// TwinCAT 3 PLC project MONETRuntime
// ProgramVersion: 3.1.4023.0
// libraries:
//   AstroBROT, * (BROT)
//   Tc2_DataExchange, * (Beckhoff Automation GmbH)
//   Tc2_Math, * (Beckhoff Automation GmbH)
//   Tc2_MC2, * (Beckhoff Automation GmbH)
//   Tc2_MC2_Drive, * (Beckhoff Automation GmbH)
//   Tc2_NC, * (Beckhoff Automation GmbH)
//   Tc2_Standard, * (Beckhoff Automation GmbH)
//   Tc2_System, * (Beckhoff Automation GmbH)
//   Tc2_Utilities, * (Beckhoff Automation GmbH)
//   Tc3_IotBase, * (Beckhoff Automation GmbH)
//   Tc3_Module, * (Beckhoff Automation GmbH)
//   VisuDialogs, * (System)
//   VisuSymbols,3.5.10.0,System
// project tree:
//   DUTs/ E_Blink.TcDUT (not stored), E_Horn.TcDUT (not stored), E_TCSCommand.TcDUT (not stored), E_TCSErrors.TcDUT (not stored), E_TelescopeMode.TcDUT (not stored), ST_InfoDataConnection.TcDUT, ST_InfoDataFB.TcDUT, ST_InfoDataGroup.TcDUT
//   / GlobalTextList.TcGTLO, PlcTask.TcTTO (not stored), Visualization Manager.TcVMO (not stored)
//   GVLs/ GVL_Hydraulics.TcGVL (not stored), GVL_Main.TcGVL, GVL_pendant_control.TcGVL (not stored), GVL_Roof.TcGVL (not stored), GVL_Safety.TcGVL, GVL_Telescope.TcGVL
//   POUs/ AzimuthElevationControl.TcPOU (not stored), CoverControl.TcPOU (not stored), DerotatorControl.TcPOU, ElevationControl.TcPOU (not stored), FocusControl.TcPOU, HydraulicsControl.TcPOU, MAIN.TcPOU, PendantControl.TcPOU, RoofControl.TcPOU (not stored), PowerMonitoring.TcPOU (not stored), SafetyHandling.TcPOU, TelescopeAuxiliary.TcPOU, TelescopeControl.TcPOU
//   POUs/FunctionBlocks/ FB_AstroClock.TcPOU (not stored), FB_Axis2.TcPOU (not stored), FB_BLINK.TcPOU (not stored), FB_ButtonEnable.TcPOU (not stored), FB_Cover.TcPOU (not stored), FB_EventLog.TcPOU (not stored), FB_Horn.TcPOU (not stored), FB_InfluxMessage.TcPOU (not stored), FB_InfoConnection.TcPOU, FB_InfoEStop.TcPOU, FB_InfoGroup.TcPOU, FB_LightTimer.TcPOU (not stored), FB_MQTTCommunication.TcPOU, FB_RFTRIG.TcPOU (not stored), FB_TimeAverage.TcPOU (not stored), FB_Timer.TcPOU (not stored), FB_TONTP.TcPOU (not stored), TelescopeAxisClass.TcPOU (not stored)
//   POUs/Functions/ CT2LST.TcPOU (not stored), F_Azimuthvelocity.TcPOU (not stored), F_DerotatorPosition2.TcPOU (not stored), F_Derotatorvelocity.TcPOU (not stored), F_Elevationvelocity.TcPOU (not stored), F_YREAL.TcPOU (not stored), NCError_TO_STRING.TcPOU (not stored), PointingModelAzimuth.TcPOU (not stored), PointingModelElevation.TcPOU (not stored), Refraction.TcPOU (not stored)
//   VISUs/ Hydraulics.TcVIS (not stored), Safety.TcVIS, Visualization.TcVIS
// real-time tasks:
//   TASK PlcTask: cycle T#10ms, priority 20, ADS port 350
// motion (NC):
//   TASK NC-Task 1 SAF: cycle T#2ms, priority 4, ADS port 501
//   TASK NC-Task 1 SVB: cycle T#10ms, priority 8, ADS port 511
//   AXIS Fokus (id 1)
//     Dynamic: AccelerationMaximum=100, DecelerationMaximum=100, Acceleration=4.5, Deceleration=4.5, Jerk=13.5
//     Velo: RefSearch=0.2, RefSync=0.2, SlowManual=0.1, FastManual=0.5, Maximum=3
//     OtherSettings: AllowMotionCmdToSlave=true, PulseDistancePos=1, PulseDistanceNeg=1
//     encoder EncType=4
//       EncPara: ScaleFactorNumerator=0.001, ScaleFactorDenominator=5, MaxCount=#x0000ffff
//         SoftEndMaxControl: Range=100
//         Inc: RefSoftSyncMask=#x0000ffff
//     drive DrvType=23
//       Analog: VeloReferenz=10.2713178, TorqueSetpointScale=10, ScaleFactorActTorque=0.2
//       TimeComp: TaskDelayCycles=1
//     controller CtrType=1
//       CtrPara: PriorControlFactor=1
//         PID: PosKp=200, CtrlOutputLimit=1
//         Observer: BandWidth=20
//   AXIS Azimuth (id 3)
//     General: UnitName=°
//     Dynamic: AccelerationMaximum=10, DecelerationMaximum=10, Acceleration=10, Deceleration=10, Jerk=4617
//     Velo: RefSearch=10.26, RefSync=10.26, SlowManual=51.3, FastManual=307.8, Fast=1026, Maximum=1026
//     OtherSettings: AllowMotionCmdToSlave=true
//     encoder EncType=8
//       EncPara: ScaleFactorNumerator=360, ScaleFactorDenominator=1048576, MaxCount=#xffffffff
//         SoftEndMinControl: Enable=true
//         SoftEndMaxControl: Enable=true, Range=450
//         Inc: RefPosition=180, RefMode=2
//     drive DrvType=9
//       DrvPara: MaxCount=#xffffffff, DriveControlDWord=#x00030100
//         Analog: VeloReferenz=1128.6, VeloScale=1.02400649589962, TorqueSetpointScale=10, ScaleFactorActTorque=0.1
//         TimeComp: TaskDelayCycles=1
//     controller CtrType=1
//       CtrPara: PriorControlFactor=1
//         PosDiffControl: Range=10
//         Observer: BandWidth=20
//   AXIS Elevation (id 4)
//     General: UnitName=°
//     Dynamic: AccelerationMaximum=10, DecelerationMaximum=10, Acceleration=10, Deceleration=10, Jerk=4617
//     Velo: RefSearch=1, RefSync=1, SlowManual=1, FastManual=3, Fast=1026, Maximum=1026
//     OtherSettings: AllowMotionCmdToSlave=true
//     encoder EncType=8
//       EncPara: ScaleFactorNumerator=360, ScaleFactorDenominator=1048576, MaxCount=#xffffffff
//         SoftEndMinControl: Enable=true
//         SoftEndMaxControl: Enable=true, Range=91
//         Inc: RefPosition=73.9885, RefMode=2
//     drive DrvType=9
//       DrvPara: MaxCount=#xffffffff, DriveControlDWord=#x00030100
//         Analog: VeloReferenz=1128.6, VeloScale=1.02400649589962, TorqueSetpointScale=10, ScaleFactorActTorque=0.1
//         TimeComp: TaskDelayCycles=1
//     controller CtrType=1
//       CtrPara: PriorControlFactor=1
//         PosDiffControl: Range=10
//         Observer: BandWidth=20
//   AXIS Derotator (id 6)
//     General: UnitName=°
//     Dynamic: Acceleration=17.5834, Deceleration=17.5834, Jerk=52.7501
//     Velo: RefSearch=0.117222517903646, RefSync=0.117222517903646, SlowManual=0.586112589518229, FastManual=3.51667553710938, Fast=11.7222517903646, Maximum=11.7223
//     OtherSettings: AllowMotionCmdToSlave=true
//     encoder EncType=8
//       EncPara: ScaleFactorNumerator=0.2, ScaleFactorDenominator=1048576, MaxCount=#xffffffff
//     drive DrvType=9
//       DrvPara: MaxCount=#xffffffff, DriveControlDWord=#x00030100
//         Analog: VeloReferenz=12.894476969401, VeloScale=1.02400649589962, TorqueSetpointScale=10, ScaleFactorActTorque=0.1
//         TimeComp: TaskDelayCycles=1
//     controller CtrType=1
//       CtrPara: PriorControlFactor=1
//         Observer: BandWidth=20
// I/O:
//   DEVICE Device 1 (EtherCAT), AmsNetId 5.131.251.159.2.1
//     Term 21 (EK1200) [EK1200-5000 EtherCAT Power supply (2A E-Bus)]
//       Term 31 (EL1004) [EL1004 4Ch. Dig. Input 24V, 3ms]
//       Temperature IN (EL3202) [EL3202 2Ch. Ana. Input PT100 (RTD)]
//       Brake AzEl (EL2004) [EL2004 4Ch. Dig. Output 24V, 0.5A] // Ch2
//       Safety Logic (EL6910) [EL6910, TwinSAFE PLC]
//       Safety IN (EL1904) [EL1904, 4 Ch. Safety Input 24V, TwinSAFE]
//         modules: Module 1 (FSOES)
//       Safety OUT (EL2904) [EL2904, 4 Ch. Safety Output 24V, 0.5A, TwinSAFE]
//         modules: Module 1 (FSOES), Module 2 (DO)
//       Hydraulics OUT (EL2008) [EL2008 8Ch. Dig. Output 24V, 0.5A] // 1: Start Oil pump. 2: Reset, 3: Start Suction pump, 4: Reset, 5: Start Oil heater, 6: Restart, 7: Brake Focus
//       Hydraulics Focus IN (EL1008) [EL1008 8Ch. Dig. Input 24V, 3ms]
//       Hydraulics IN2 (EL1008) [EL1008 8Ch. Dig. Input 24V, 3ms]
//       Focus Motor (EL7342) [EL7342 2Ch. DC motor output stage (50V, 3.5A)]
//       Mirror Temperature IN (EL3164) [EL3164 4Ch. Ana. Input 0-10V]
//       Power Analysis (EL3483) [EL3483 3Ch. Mains Monitoring]
//       Power (EL9410) [EL9410 E-Bus Power Supplier  (Diagnostics)]
//       Mirror Cover OUT1 (EL2004) [EL2004 4Ch. Dig. Output 24V, 0.5A]
//       Mirror Cover OUT2 (EL2004) [EL2004 4Ch. Dig. Output 24V, 0.5A]
//       Mirror Cover IN (EL1008) [EL1008 8Ch. Dig. Input 24V, 3ms]
//       Front Panel IN (EL1008) [EL1008 8Ch. Dig. Input 24V, 3ms]
//       Front Panel OUT (EL2004) [EL2004 4Ch. Dig. Output 24V, 0.5A]
//       Pendant Control IN (EL1008) [EL1008 8Ch. Dig. Input 24V, 3ms]
//       Pendant Control IN2 (EL1008) [EL1008 8Ch. Dig. Input 24V, 3ms]
//       Pendant Control OUT (EL2008) [EL2008 8Ch. Dig. Output 24V, 0.5A]
//       Cabinet OUT (EL2004) [EL2004 4Ch. Dig. Output 24V, 0.5A]
//       Term 48 (EL9011) [EL9011 End Terminal]
//   DEVICE Device 5 (EtherCAT), AmsNetId 5.131.251.159.6.1
//     Azimuth (AX5125-0000-0214) [AX5125-0000-0214 EtherCAT Drive (SoE, 1 Ch.)]
//       Term 2 (AX5805) [AX5805 (Safety Drive Option)]
//         modules: Module 1 (Safety Process Data, 1 axis), Module 2 (Standard Process Data, 1 axis)
//       Term 7 (EL9011) [EL9011 End Terminal]
//     Elevation (AX5125-0000-0214) [AX5125-0000-0214 EtherCAT Drive (SoE, 1 Ch.)]
//       Term 4 (AX5805) [AX5805 (Safety Drive Option)]
//         modules: Module 1 (Safety Process Data, 1 axis), Module 2 (Standard Process Data, 1 axis)
//       Term 8 (EL9011) [EL9011 End Terminal]
//     Derotator (AX5206-0000-0214) [AX5206-0000-0214 EtherCAT Drive (SoE, 2 Ch.)]
//       Term 6 (AX5805) [AX5805 (Safety Drive Option)]
//         modules: Module 1 (Safety Process Data, 2 axis), Module 2 (Standard Process Data, 2 axis)
//       Term 9 (EL9011) [EL9011 End Terminal]
// variable links:
//   Device 1 (EtherCAT) <-> Device 1 (EtherCAT)/Term 21 (EK1200)/Safety IN (EL1904)
//     Term 21 (EK1200)/Safety Logic (EL6910)/ConnectionInputs/Message_7 TxPDO <-> Module 1 (FSOES)/RxPDO/FSOE
//     Term 21 (EK1200)/Safety Logic (EL6910)/ConnectionOutputs/Message_7 RxPDO <-> Module 1 (FSOES)/TxPDO/FSOE
//   Device 1 (EtherCAT) <-> Device 1 (EtherCAT)/Term 21 (EK1200)/Safety Logic (EL6910)
//     Term 21 (EK1200)/Safety OUT (EL2904)/Module 1 (FSOES)/TxPDO/FSOE <-> ConnectionOutputs/Message_8 RxPDO
//   Device 1 (EtherCAT) <-> Device 1 (EtherCAT)/Term 21 (EK1200)/Safety OUT (EL2904)
//     Term 21 (EK1200)/Safety Logic (EL6910)/ConnectionInputs/Message_8 TxPDO <-> Module 1 (FSOES)/RxPDO/FSOE
//   Device 1 (EtherCAT) <-> Device 5 (EtherCAT)/Azimuth (AX5125-0000-0214)/Term 2 (AX5805)
//     Term 21 (EK1200)/Safety Logic (EL6910)/ConnectionInputs/Message_5 TxPDO <-> Module 1 (Safety Process Data, 1 axis)/Outputs (Controlword)/FSOE
//     Term 21 (EK1200)/Safety Logic (EL6910)/ConnectionOutputs/Message_5 RxPDO <-> Module 1 (Safety Process Data, 1 axis)/Inputs (Statusword)/FSOE
//   Device 1 (EtherCAT) <-> Device 5 (EtherCAT)/Derotator (AX5206-0000-0214)/Term 6 (AX5805)
//     Term 21 (EK1200)/Safety Logic (EL6910)/ConnectionOutputs/Message_17 RxPDO <-> Module 1 (Safety Process Data, 2 axis)/Inputs (Statusword)/FSOE
//   Device 5 (EtherCAT) <-> Device 1 (EtherCAT)/Term 21 (EK1200)/Safety Logic (EL6910)
//     Derotator (AX5206-0000-0214)/Term 6 (AX5805)/Module 1 (Safety Process Data, 2 axis)/Outputs (Controlword)/FSOE <-> ConnectionInputs/Message_17 TxPDO
//     Elevation (AX5125-0000-0214)/Term 4 (AX5805)/Module 1 (Safety Process Data, 1 axis)/Inputs (Statusword)/FSOE <-> ConnectionOutputs/Message_6 RxPDO
//     Elevation (AX5125-0000-0214)/Term 4 (AX5805)/Module 1 (Safety Process Data, 1 axis)/Outputs (Controlword)/FSOE <-> ConnectionInputs/Message_6 TxPDO
//   NC-Task 1 SAF/Axes/Azimuth <-> Device 5 (EtherCAT)/Azimuth (AX5125-0000-0214)
//     Drive/Inputs/In/nDataIn1 <-> AT/Following distance
//     Drive/Inputs/In/nDcOutputTime <-> InfoData/DcOutputShift
//     Drive/Inputs/In/nState1 <-> AT/Drive status word @bit 8
//     Drive/Inputs/In/nState2 <-> AT/Drive status word
//     Drive/Inputs/In/nState4 @bit 1 <-> WcState/InputToggle
//     Drive/Inputs/In/nState4 <-> WcState/WcState
//     Drive/Outputs/Out/nCtrl1 <-> MDT/Master control word @bit 8
//     Drive/Outputs/Out/nDataOut1 <-> MDT/Position command value
//     Enc/Inputs/In/nDataIn1 <-> AT/Position feedback 1 value
//     Enc/Inputs/In/nDataIn3 <-> AT/Probe value 1 positive edge
//     Enc/Inputs/In/nDataIn4 <-> AT/Probe value 1 negative edge
//     Enc/Inputs/In/nDcInputTime <-> InfoData/DcInputShift
//     Enc/Inputs/In/nState4 @bit 1 <-> WcState/InputToggle
//     Enc/Inputs/In/nState4 <-> WcState/WcState
//     Enc/Inputs/In/nState5 <-> AT/Probe 1 positive latched
//     Enc/Inputs/In/nState6 <-> AT/Probe 1 negative latched
//     Enc/Outputs/Out/nCtrl5 <-> MDT/Probe 1 enable
//   NC-Task 1 SAF/Axes/Derotator <-> Device 5 (EtherCAT)/Derotator (AX5206-0000-0214)
//     Drive/Inputs/In/nDataIn1 <-> AT 1/Following distance
//     Drive/Inputs/In/nDcOutputTime <-> InfoData/DcOutputShift
//     Drive/Inputs/In/nState1 <-> AT 1/Drive status word @bit 8
//     Drive/Inputs/In/nState2 <-> AT 1/Drive status word
//     Drive/Inputs/In/nState4 @bit 1 <-> WcState/InputToggle
//     Drive/Inputs/In/nState4 <-> WcState/WcState
//     Drive/Outputs/Out/nCtrl1 <-> MDT 1/Master control word @bit 8
//     Drive/Outputs/Out/nDataOut1 <-> MDT 1/Position command value
//     Enc/Inputs/In/nDataIn1 <-> AT 1/Position feedback 1 value
//     Enc/Inputs/In/nDcInputTime <-> InfoData/DcInputShift
//     Enc/Inputs/In/nState4 @bit 1 <-> WcState/InputToggle
//     Enc/Inputs/In/nState4 <-> WcState/WcState
//   NC-Task 1 SAF/Axes/Elevation <-> Device 5 (EtherCAT)/Elevation (AX5125-0000-0214)
//     Drive/Inputs/In/nDataIn1 <-> AT/Following distance
//     Drive/Inputs/In/nDcOutputTime <-> InfoData/DcOutputShift
//     Drive/Inputs/In/nState1 <-> AT/Drive status word @bit 8
//     Drive/Inputs/In/nState2 <-> AT/Drive status word
//     Drive/Inputs/In/nState4 @bit 1 <-> WcState/InputToggle
//     Drive/Inputs/In/nState4 <-> WcState/WcState
//     Drive/Outputs/Out/nCtrl1 <-> MDT/Master control word @bit 8
//     Drive/Outputs/Out/nDataOut1 <-> MDT/Position command value
//     Enc/Inputs/In/nDataIn1 <-> AT/Position feedback 1 value
//     Enc/Inputs/In/nDataIn3 <-> AT/Probe value 1 positive edge
//     Enc/Inputs/In/nDataIn4 <-> AT/Probe value 1 negative edge
//     Enc/Inputs/In/nDcInputTime <-> InfoData/DcInputShift
//     Enc/Inputs/In/nState4 @bit 1 <-> WcState/InputToggle
//     Enc/Inputs/In/nState4 <-> WcState/WcState
//     Enc/Inputs/In/nState5 <-> AT/Probe 1 positive latched
//     Enc/Inputs/In/nState6 <-> AT/Probe 1 negative latched
//     Enc/Outputs/Out/nCtrl5 <-> MDT/Probe 1 enable
//   NC-Task 1 SAF/Axes/Fokus <-> Device 1 (EtherCAT)/Term 21 (EK1200)/Focus Motor (EL7342)
//     Drive/Inputs/In/nDcOutputTime <-> InfoData/DcOutputShift
//     Drive/Inputs/In/nState1 @bit 3 <-> DCM Status Channel 1/Status/Error
//     Drive/Inputs/In/nState1 @bit 5 <-> DCM Status Channel 1/Status/Moving negative
//     Drive/Inputs/In/nState1 @bit 4 <-> DCM Status Channel 1/Status/Moving positive
//     Drive/Inputs/In/nState1 @bit 1 <-> DCM Status Channel 1/Status/Ready
//     Drive/Inputs/In/nState1 <-> DCM Status Channel 1/Status/Ready to enable
//     Drive/Inputs/In/nState1 @bit 6 <-> DCM Status Channel 1/Status/Torque reduced
//     Drive/Inputs/In/nState1 @bit 2 <-> DCM Status Channel 1/Status/Warning
//     Drive/Inputs/In/nState2 @bit 3 <-> DCM Status Channel 1/Status/Digital input 1
//     Drive/Inputs/In/nState2 @bit 4 <-> DCM Status Channel 1/Status/Digital input 2
//     Drive/Inputs/In/nState2 @bit 5 <-> DCM Status Channel 1/Status/Sync error
//     Drive/Inputs/In/nState2 @bit 7 <-> DCM Status Channel 1/Status/TxPDO Toggle
//     Drive/Inputs/In/nState4 @bit 1 <-> WcState/InputToggle
//     Drive/Inputs/In/nState4 <-> WcState/WcState
//     Drive/Outputs/Out/nCtrl1 <-> DCM Control Channel 1/Control/Enable
//     Drive/Outputs/Out/nCtrl1 @bit 2 <-> DCM Control Channel 1/Control/Reduce torque
//     Drive/Outputs/Out/nCtrl1 @bit 1 <-> DCM Control Channel 1/Control/Reset
//     Drive/Outputs/Out/nCtrl1 @bit 3 <-> DCM Control Channel 1/Control/Threshold active
//     Drive/Outputs/Out/nDataOut2[0] <-> DCM Velocity Channel 1/Velocity
//     Enc/Inputs/In/nDataIn1[0] <-> ENC Status compact Channel 1/Counter value
//     Enc/Inputs/In/nDataIn2[0] <-> ENC Status compact Channel 1/Latch value
//     Enc/Inputs/In/nDcInputTime <-> InfoData/DcInputShift
//     Enc/Inputs/In/nState1 @bit 4 <-> ENC Status compact Channel 1/Status/Counter overflow
//     Enc/Inputs/In/nState1 @bit 3 <-> ENC Status compact Channel 1/Status/Counter underflow
//     Enc/Inputs/In/nState1 @bit 7 <-> ENC Status compact Channel 1/Status/Extrapolation stall
//     Enc/Inputs/In/nState1 @bit 1 <-> ENC Status compact Channel 1/Status/Latch extern valid
//     Enc/Inputs/In/nState1 @bit 2 <-> ENC Status compact Channel 1/Status/Set counter done
//     Enc/Inputs/In/nState2 @bit 4 <-> ENC Status compact Channel 1/Status/Status of extern latch
//     Enc/Inputs/In/nState2 <-> ENC Status compact Channel 1/Status/Status of input A
//     Enc/Inputs/In/nState2 @bit 1 <-> ENC Status compact Channel 1/Status/Status of input B
//     Enc/Inputs/In/nState2 @bit 5 <-> ENC Status compact Channel 1/Status/Sync error
//     Enc/Inputs/In/nState2 @bit 7 <-> ENC Status compact Channel 1/Status/TxPDO Toggle
//     Enc/Inputs/In/nState4 @bit 1 <-> WcState/InputToggle
//     Enc/Inputs/In/nState4 <-> WcState/WcState
//     Enc/Outputs/Out/nCtrl1 @bit 3 <-> ENC Control compact Channel 1/Control/Enable latch extern on negative edge
//     Enc/Outputs/Out/nCtrl1 @bit 1 <-> ENC Control compact Channel 1/Control/Enable latch extern on positive edge
//     Enc/Outputs/Out/nCtrl1 @bit 2 <-> ENC Control compact Channel 1/Control/Set counter
//     Enc/Outputs/Out/nDataOut1[0] <-> ENC Control compact Channel 1/Set counter value
//   MONETRuntime/MONETRuntime Instance <-> Device 1 (EtherCAT)/Term 21 (EK1200)/Brake AzEl (EL2004)
//     PlcTask Outputs/GVL_Telescope.brake_azimuth_eve <-> Channel 2/GVL_Telescope.brake_azimuth_eve
//   MONETRuntime/MONETRuntime Instance <-> Device 1 (EtherCAT)/Term 21 (EK1200)/Front Panel IN (EL1008)
//     PlcTask Inputs/GVL_Main.brake_clearing <-> Channel 5/GVL_Main.key_brake_clearing
//     PlcTask Inputs/GVL_Main.key_switch_remote <-> Channel 4/GVL_Main.key_switch_remote
//     PlcTask Inputs/GVL_Main.reset_switch <-> Channel 3/GVL_Main.reset_switch
//     PlcTask Inputs/GVL_Main.start_switch <-> Channel 1/GVL_Main.start_switch
//     PlcTask Inputs/GVL_Main.stop_switch <-> Channel 2/GVL_Main.stop_switch
//   MONETRuntime/MONETRuntime Instance <-> Device 1 (EtherCAT)/Term 21 (EK1200)/Front Panel OUT (EL2004)
//     PlcTask Outputs/GVL_Main.lamp_error <-> Channel 3/GVL_Main.lamp_error
//     PlcTask Outputs/GVL_Main.lamp_on_manual <-> Channel 2/GVL_Main.lamp_ready
//     PlcTask Outputs/GVL_Main.lamp_power <-> Channel 1/GVL_Main.lamp_power
//   MONETRuntime/MONETRuntime Instance <-> Device 1 (EtherCAT)/Term 21 (EK1200)/Hydraulics Focus IN (EL1008)
//     PlcTask Inputs/GVL_Hydraulics.pump_running <-> Channel 1/GVL_Hydraulics.pump_running
//     PlcTask Inputs/GVL_Hydraulics.suction_running <-> Channel 2/GVL_Hydraulics.suction_running
//     PlcTask Inputs/GVL_Telescope.focus_limit_far <-> Channel 5/GVL_Telescope.focus_limit_far
//     PlcTask Inputs/GVL_Telescope.focus_limit_near <-> Channel 4/GVL_Telescope.focus_limit_near
//   MONETRuntime/MONETRuntime Instance <-> Device 1 (EtherCAT)/Term 21 (EK1200)/Hydraulics IN2 (EL1008)
//     PlcTask Inputs/GVL_Hydraulics.oil_high <-> Channel 2/GVL_Hydraulics.oil_high
//     PlcTask Inputs/GVL_Hydraulics.oil_low <-> Channel 1/GVL_Hydraulics.oil_low
//     PlcTask Inputs/GVL_Hydraulics.oil_overtemperature <-> Channel 4/GVL_Hydraulics.oil_overtemperature
//     PlcTask Inputs/GVL_Hydraulics.oil_pressure_OK <-> Channel 3/GVL_Hydraulics.pressure_OK
//     PlcTask Inputs/GVL_Hydraulics.oil_reserve <-> Channel 8/GVL_Hydraulics.oil_reserve
//     PlcTask Inputs/GVL_Hydraulics.oil_undertemperature <-> Channel 5/GVL_Hydraulics.oil_undertemperature
//     PlcTask Inputs/GVL_Hydraulics.oilfilter_dirty <-> Channel 6/GVL_Hydraulics.oilfilter_dirty
//     PlcTask Inputs/GVL_Hydraulics.oilpan_maximum <-> Channel 7/GVL_Hydraulics.oilpan_maximum
//   MONETRuntime/MONETRuntime Instance <-> Device 1 (EtherCAT)/Term 21 (EK1200)/Hydraulics OUT (EL2008)
//     PlcTask Outputs/GVL_Hydraulics.oil_pump_enable <-> Channel 1/GVL_Hydraulics.oil_pump_enable
//     PlcTask Outputs/GVL_Hydraulics.oil_suction_enable <-> Channel 3/GVL_Hydraulics.oil_suction_enable
//     PlcTask Outputs/GVL_Telescope.focus_unlock <-> Channel 7/GVL_Telescope.focus_unlock
//   MONETRuntime/MONETRuntime Instance <-> Device 1 (EtherCAT)/Term 21 (EK1200)/Mirror Cover IN (EL1008)
//     PlcTask Inputs/GVL_Telescope.cover1_closed <-> Channel 2/GVL_Telescope.cover1_closed
//     PlcTask Inputs/GVL_Telescope.cover2_closed <-> Channel 4/GVL_Telescope.cover2_closed
//     PlcTask Inputs/GVL_Telescope.cover3_closed <-> Channel 6/GVL_Telescope.cover3_closed
//     PlcTask Inputs/GVL_Telescope.cover1_open <-> Channel 1/GVL_Telescope.cover1_open
//     PlcTask Inputs/GVL_Telescope.cover2_open <-> Channel 3/GVL_Telescope.cover2_open
//     PlcTask Inputs/GVL_Telescope.cover3_open <-> Channel 5/GVL_Telescope.cover3_open
//   MONETRuntime/MONETRuntime Instance <-> Device 1 (EtherCAT)/Term 21 (EK1200)/Mirror Cover OUT1 (EL2004)
//     PlcTask Outputs/GVL_Telescope.close_cover1 <-> Channel 2/GVL_Telescope.close_cover1
//     PlcTask Outputs/GVL_Telescope.close_cover2 <-> Channel 4/GVL_Telescope.close_cover2
//     PlcTask Outputs/GVL_Telescope.open_cover1 <-> Channel 1/GVL_Telescope.open_cover1
//     PlcTask Outputs/GVL_Telescope.open_cover2 <-> Channel 3/GVL_Telescope.open_cover2
//   MONETRuntime/MONETRuntime Instance <-> Device 1 (EtherCAT)/Term 21 (EK1200)/Mirror Cover OUT2 (EL2004)
//     PlcTask Outputs/GVL_Telescope.close_cover3 <-> Channel 2/GVL_Telescope.close_cover3
//     PlcTask Outputs/GVL_Telescope.open_cover3 <-> Channel 1/GVL_Telescope.open_cover3
//   MONETRuntime/MONETRuntime Instance <-> Device 1 (EtherCAT)/Term 21 (EK1200)/Mirror Temperature IN (EL3164)
//     PlcTask Inputs/GVL_Telescope.temperature_mirror1 <-> AI Standard Channel 2/Value
//     PlcTask Inputs/GVL_Telescope.temperature_mirror2 <-> AI Standard Channel 1/Value
//   MONETRuntime/MONETRuntime Instance <-> Device 1 (EtherCAT)/Term 21 (EK1200)/Pendant Control IN (EL1008)
//     PlcTask Inputs/GVL_pendant_control.BCD1 <-> Channel 1/GVL_pendant_control.BCD0
//     PlcTask Inputs/GVL_pendant_control.BCD2 <-> Channel 2/GVL_pendant_control.BCD2
//     PlcTask Inputs/GVL_pendant_control.BCD4 <-> Channel 3/GVL_pendant_control.BCD4
//     PlcTask Inputs/GVL_pendant_control.BCD8 <-> Channel 4/GVL_pendant_control.BCD8
//     PlcTask Inputs/GVL_pendant_control.direction_down <-> Channel 7/GVL_pendant_control.direction_down
//     PlcTask Inputs/GVL_pendant_control.direction_up <-> Channel 6/GVL_pendant_control.direction_up
//     PlcTask Inputs/GVL_pendant_control.key_switch <-> Channel 8/GVL_pendant_control.key_switch
//     PlcTask Inputs/GVL_pendant_control.reset_switch <-> Channel 5/GVL_pendant_control.reset_switch
//   MONETRuntime/MONETRuntime Instance <-> Device 1 (EtherCAT)/Term 21 (EK1200)/Pendant Control IN2 (EL1008)
//     PlcTask Inputs/GVL_pendant_control.direction_left <-> Channel 2/GVL_pendant_control.direction_left
//     PlcTask Inputs/GVL_pendant_control.direction_right <-> Channel 3/GVL_pendant_control.direction_right
//     PlcTask Inputs/GVL_pendant_control.start_switch <-> Channel 1/GVL_pendant_control.start_switch
//   MONETRuntime/MONETRuntime Instance <-> Device 1 (EtherCAT)/Term 21 (EK1200)/Pendant Control OUT (EL2008)
//     PlcTask Outputs/GVL_pendant_control.lamp_down <-> Channel 2/GVL_pendant_control.lamp_down
//     PlcTask Outputs/GVL_pendant_control.lamp_error <-> Channel 5/GVL_pendant_control.lamp_error
//     PlcTask Outputs/GVL_pendant_control.lamp_left <-> Channel 4/GVL_pendant_control.lamp_left
//     PlcTask Outputs/GVL_pendant_control.lamp_right <-> Channel 3/GVL_pendant_control.lamp_right
//     PlcTask Outputs/GVL_pendant_control.lamp_up <-> Channel 1/GVL_pendant_control.lamp_up
//   MONETRuntime/MONETRuntime Instance <-> Device 1 (EtherCAT)/Term 21 (EK1200)/Safety Logic (EL6910)
//     PlcTask Inputs/GVL_Telescope.Azimuth_sto <-> StandardInputs/Standard Out Var 18
//     PlcTask Inputs/GVL_Telescope.Derotator_sto <-> StandardInputs/Standard Out Var 20
//     PlcTask Inputs/GVL_Telescope.Elevation_sto <-> StandardInputs/Standard Out Var 19
//     PlcTask Inputs/SafetyHandling.stInfoEStop1 <-> Function Block Info Data/TwinSafeGroup1.Network1.FBEstop1 Info Data
//     PlcTask Inputs/SafetyHandling.stInfoGroup1 <-> TwinSAFE Group Info Data/TwinSafeGroup1 Info Data
//     PlcTask Inputs/SafetyHandling.stInfoSafetyIn <-> Connection Info Data/Message_8 Info Data
//     PlcTask Inputs/SafetyHandling.stInfoSafetyOut <-> Connection Info Data/Message_7 Info Data
//     PlcTask Outputs/GVL_Safety.ErrAck <-> StandardOutputs/Standard In Var 1
//     PlcTask Outputs/GVL_Safety.Reset_STO_Azimuth <-> StandardOutputs/Standard In Var 25
//     PlcTask Outputs/GVL_Safety.Reset_STO_Derotator <-> StandardOutputs/Standard In Var 22
//     PlcTask Outputs/GVL_Safety.Reset_STO_Elevation <-> StandardOutputs/Standard In Var 26
//     PlcTask Outputs/GVL_Safety.Restart <-> StandardOutputs/Standard In Var 3
//     PlcTask Outputs/GVL_Safety.Run <-> StandardOutputs/Standard In Var 2
//   MONETRuntime/MONETRuntime Instance <-> Device 1 (EtherCAT)/Term 21 (EK1200)/Temperature IN (EL3202)
//     PlcTask Inputs/GVL_Main.main_cabinet_temperature <-> RTD Inputs Channel 1/Value

// ---- DUTs/ST_InfoDataConnection.TcDUT
TYPE ST_InfoDataConnection :
STRUCT
	usiMapState	:USINT;
	usiMapDiag	:USINT;
	bySignal	:BYTE;
END_STRUCT
END_TYPE

// ---- DUTs/ST_InfoDataFB.TcDUT
TYPE ST_InfoDataFB :
STRUCT
	usiMapState	:USINT;
	uiMapDiag	:USINT;
	usiDummy	:USINT;
END_STRUCT
END_TYPE

// ---- DUTs/ST_InfoDataGroup.TcDUT
TYPE ST_InfoDataGroup :
STRUCT
	usiMapState	:USINT;
	usiMapDiag	:USINT;	
END_STRUCT
END_TYPE

// ---- GVLs/GVL_Main.TcGVL
{attribute 'qualified_only'}
//TODO update to current RoboTel IOs
VAR_GLOBAL
	//DIN1 0.0
	//phase_available		AT%I*: BOOL;
	//not implemented on RoboTel
	//key_switch			AT%I*: BOOL;
	//DIN3 0.2
	key_switch_remote	AT%I*: BOOL;
	//DIN4 0.3
	start_switch		AT%I*: BOOL;
	//DIN5 0.4
	stop_switch			AT%I*: BOOL;
	//DIN8 0.7
	reset_switch		AT%I*: BOOL;
	
	//BT1
	main_cabinet_temperature	AT%I*: INT;
	//DIN15 1.6
	brake_clearing		AT%I*: BOOL;
	
	//DOUT1 0.0
	lamp_power			AT%Q*: BOOL;
	//DOUT2 0.1
	lamp_on_manual			AT%Q*: BOOL;
	//DOUT3 0.2
	lamp_error			AT%Q*: BOOL;
	
	isRoboTel:		BOOL;
	(*
	NeutralCurrentGuardWarning		AT%I*:	BOOL;
	NeutralCurrentGuarError			AT%I*:	BOOL;
	ActivePowerGuardWarning			AT%I*:	BOOL;
	ActivePowerGuardError			AT%I*:	BOOL;
	ApparentPowerGuardWarning		AT%I*:	BOOL;
	ApparentPowerGuardError			AT%I*:	BOOL;
	*)
	//ActivePower						AT%I*:	REAL;
	//ActiveEnergy					AT%I*:	LINT;
	//NeutralLineCurrent				AT%I*:	REAL;
END_VAR

// ---- GVLs/GVL_Safety.TcGVL
{attribute 'qualified_only'}
VAR_GLOBAL
	// Safety Error Condition
	Error		AT%I*:	BOOL;
	// Run/Stop Safety
	Run			AT%Q*:	BOOL;
	// Restart Safety
	Restart		AT%Q*:	BOOL;
	// Error Acknowledgement 
	ErrAck		AT%Q*:	BOOL;
	// Stop signal coming from Safety
	// Stop		AT%I*:	BOOL;
	// state variable
	State		AT%I*:	USINT;
	
	Reset_STO_Azimuth		AT%Q*: BOOL;
	Reset_STO_Elevation		AT%Q*: BOOL;
	Reset_STO_Derotator		AT%Q*: BOOL;
END_VAR

// ---- GVLs/GVL_Telescope.TcGVL
{attribute 'qualified_only'}
VAR_GLOBAL
	// BT9 mirror
	temperature_mirror2		AT%I*: INT;
	// BT10
	temperature_mirror1		AT%I*: INT;

	//DOUT6 0.5
	brake_azimuth_eve	AT%Q*: BOOL;
	
	// DIN28 3.3 (absolute)
	azimut_limit_switch	AT%I*: BOOL;
	// DIN29 3.4
	focus_limit_near	AT%I*: BOOL;
	// DIN30 3.5
	focus_limit_far		AT%I*: BOOL;
	
	// DIN33 4.0
	cover1_open		AT%I*: BOOL;
	// DIN34 4.1
	cover1_closed	AT%I*: BOOL;
	// DIN35 4.2
	cover2_open		AT%I*: BOOL;
	// DIN36 4.3
	cover2_closed	AT%I*: BOOL;
	// DIN37 4.4
	cover3_open		AT%I*: BOOL;
	// DIN38 4.5
	cover3_closed	AT%I*: BOOL;

	//DOUT14 1.5
	focus_unlock		AT%Q*: BOOL;
	//Horn 4.7
	horn			AT%Q*: BOOL;
	
	// digitale inputs der Endlagen
	Derotator_inputs		AT%I*: WORD;
	// diagnostic number
	Derotator_diagnostic	AT%I*: UDINT;
	// derotator torque feedback
	Derotator_torque		AT%I*: INT;
	// STO
	Derotator_sto			AT%I*: BOOL;
	
	// digital inputs for limit switches
	Elevation_inputs		AT%I*: WORD;
	// diagnostic number
	Elevation_diagnostic	AT%I*: UDINT;
	// torque feedback
	Elevation_torque		AT%I*: INT;
	// STO
	Elevation_sto			AT%I*: BOOL;
	
	// digital inputs for limit switches
	Azimuth_inputs			AT%I*: WORD;
	// diagnostic number
	Azimuth_diagnostic		AT%I*: UDINT;
	// torque feedback
	Azimuth_torque			AT%I*: INT;
	// STO
	Azimuth_sto				AT%I*: BOOL;	
	
	// Zyklisches Interface zwischen NC und Achse
	AzimuthAxisRef: 	AXIS_REF;
	ElevationAxisRef: 	AXIS_REF;
	DerotatorAxisRef: 	AXIS_REF;
 	// Motor1 Channel 1
	FocusAxisRef:		AXIS_REF;
	
	//nasmyth_left	AT%Q*: BOOL;
	//nasmyth_right	AT%Q*: BOOL;
	open_cover1		AT%Q*: BOOL;
	close_cover1	AT%Q*: BOOL;
	open_cover2		AT%Q*: BOOL;
	close_cover2	AT%Q*: BOOL;
	open_cover3		AT%Q*: BOOL;
	close_cover3	AT%Q*: BOOL;
	
	
END_VAR

// ---- POUs/DerotatorControl.TcPOU
PROGRAM DerotatorControl
VAR_INPUT
	// enable the derotator
	enable:		BOOL;
	// reset an error
	reset:		BOOL;
	// decrease derotator angle
	left:		BOOL;
	// increase derotator angle
	right:		BOOL;
	// set the absolute position
	position:	LREAL;
	// derotator velocity
	Velocity:	LREAL := 10.0;
	// move to given position
	MoveAxis: 	BOOL;
	// calibrate the axis
	HomeAxis:	BOOL;
	// tracking flag
	Tracking:	BOOL;
	// stop the Axis
	StopAxis:	BOOL;
	// diagnostic error code reset
	bSoEReset: 			BOOL;
END_VAR
VAR_OUTPUT
	// error flag
	Error:				BOOL;
	// nc error id
	ErrorID:			UDINT;
	// actual position of the derotator
	actual_position:	LREAL;
	// calibrated flag
	Calibrated:			BOOL;
	// axis ready flag
	Ready:				BOOL;
	// position to move the axis to
	slewtime: 			LREAL;
END_VAR
VAR
	// trigger for the torque error
	TorqueError:		TON := (PT := T#3S);
	// axis function block
	DerotatorAxis:		FB_Axis2;
	
	DerotatorEvent:		FB_EventLog;
	// torque warning event
	TorqueWarning:		FB_EventLog;
	// torque calibration event
	CalibrationEvent:	FB_EventLog;
	// diagnostic low-level event
	DerotatorDiagnosticEvent: FB_EventLog;
	// percentage of the derotator torque
	derotator_torque:	REAL;
	// read slewtime
	ReadParameter:		MC_ReadParameter;
	fbSoEReset: 		FB_SoEReset;
	DiagnosticError:	BOOL;
END_VAR
VAR CONSTANT
	// current position of the calibration cam. Apply an offset here if necessary
	calibration_position:	LREAL := 438.4623; // calibration in positive direction (was 460.0)
END_VAR

(*
Selection 6
Homing in Endlage:

https://infosys.beckhoff.com/index.php?content=../content/1031/ax5000_usermanual/html/ax5000_homing_hardware_end_position.htm&id=12221
NC-Interface:
PlcToNc-Achsinterface, Bit 8 namens AcceptBlockedDriveSignal im nDeCtrlDWord

SPS-Interface:
TcNc-Lib, siehe SPS-Funktion AxisSetAcceptBlockedDriveSignal in der TwinCAT  PLC Library: NC.
*)

position := LIMIT(-70, position, 380);

IF enable AND NOT DerotatorAxis.Calibrated THEN
	HomeAxis := TRUE;
END_IF

IF DerotatorAxis.Calibrated THEN
	HomeAxis := FALSE;
	Calibrated := DerotatorAxis.Calibrated;
END_IF
	
IF HomeAxis THEN
	position := calibration_position;
END_IF

DeRotatorAxis(
	enable := 			enable,
	Reset := 			Reset,
	MoveAxis :=			MoveAxis,
	HomeAxis :=			HomeAxis,
	StopAxis :=			StopAxis,
	HomingMode :=		MC_ForceCalibration,
	Position := 		position, 
	Velocity :=			Velocity,
	Enable_Positive := 	NOT GVL_Telescope.Derotator_inputs.0,
	Enable_Negative := 	NOT GVL_Telescope.Derotator_inputs.1,
	Jog_Forward := 		right,
	Jog_Backwards := 	left,
	bCalibrationCam :=	GVL_Telescope.Derotator_inputs.0,
	isModuloAxis :=		FALSE,
	Tracking :=			Tracking,
	ActualPosition => 	actual_position,
	Error => 			Error,
	ErrorID => 			ErrorID,
	AxisRef :=			GVL_Telescope.DerotatorAxisRef);
	
IF DeRotatorAxis.MoveDone OR Reset OR Error THEN
	MoveAxis := FALSE;
END_IF

IF DeRotatorAxis.HomeDone OR Reset OR Error THEN
	HomeAxis := FALSE;
END_IF
	
IF DeRotatorAxis.ResetDone THEN
	reset := FALSE;
END_IF

IF DeRotatorAxis.StopDone THEN
	StopAxis := FALSE;
END_IF

DiagnosticError := FALSE;
IF GVL_Telescope.Derotator_diagnostic < 16#D012 AND GVL_Telescope.Derotator_diagnostic > 16#D014 THEN
	DiagnosticError := TRUE;
	ErrorID := GVL_Telescope.Derotator_diagnostic;
	bSoeReset := reset;
END_IF

Ready := DeRotatorAxis.Ready;

ReadParameter(	Axis := GVL_Telescope.DerotatorAxisRef, 
				Enable := DeRotatorAxis.InMotion, 
				ParameterNumber := MC_AxisParameter.AxisRemainingTimeToGo, 
				ReadMode := E_ReadMode.READMODE_CYCLIC);
				
IF ReadParameter.Valid THEN
	slewtime := ReadParameter.Value;
END_IF

IF bSoEReset THEN
	fbSoEReset(
		Axis := GVL_Telescope.DerotatorAxisRef,
		Execute := TRUE,
		Timeout := DEFAULT_ADS_TIMEOUT);
 	IF NOT fbSoEReset.Busy THEN
		fbSoEReset(Axis := GVL_Telescope.DerotatorAxisRef, Execute := FALSE);
		bSoEReset := FALSE;
		Reset := TRUE;
	END_IF
END_IF

derotator_torque := GVL_Telescope.Derotator_torque / 10.0;

TorqueError(IN := ABS(derotator_torque) > 12.0);

DerotatorEvent(	
	Trigger := 		Error, 
	Level := 		ADSLOG_MSGTYPE_ERROR,
	FormatString :=	'Derotator Axis Error: %s',
	OnMessage := 	NCError_TO_STRING(ErrorID),
	OffMEssage := 	'OK',
	OffLevel := 	ADSLOG_MSGTYPE_HINT);
	
DerotatorDiagnosticEvent(	
	Trigger := 		DiagnosticError, 
	Level := 		ADSLOG_MSGTYPE_ERROR,
	FormatString :=	'Derotator Axis Diagnostic Error: %s',
	OnMessage := 	NCError_TO_STRING(GVL_Telescope.Derotator_diagnostic));
	
TorqueWarning(	
	Trigger := 		TorqueError.Q, 
	Level := 		ADSLOG_MSGTYPE_WARN,
	FormatString :=	'%s',
	OnMessage := 	'Derotator torque is high.');

CalibrationEvent(	
	Trigger := 		Calibrated, 
	Level := 		ADSLOG_MSGTYPE_HINT,
	OnMessage := 	'Derotator is calibrated.');

END_PROGRAM

// ---- POUs/FocusControl.TcPOU
PROGRAM FocusControl
VAR_INPUT
	// enable the axis
	enable: BOOL;
	// Move M2 closer to M1
	inward: 	BOOL;
	// Move M2 away from M1
	outward: 	BOOL;	
	// reset the axis(-error)
	reset: 		BOOL;
	// move the axis to new position
	MoveAxis:	BOOL;
	// calibrate the focus axis
	HomeAxis:	BOOL;
	// focus position in millimeters
	position: 		LREAL;
END_VAR

VAR_OUTPUT
	// true if absolute calibration
	Calibrated:	BOOL;
	// true if error
	Error: 		BOOL;
	// ID of NC axis error
	ErrorID:	UDINT;
	// ready signal = drive ready + standstill
	Ready:	BOOL;
END_VAR

VAR
	FocusDelay:			TON;
	BrakeDelay:			TON;
	FocusAxis:			FB_Axis2;
	actual_position:	LREAL;
	// manual override to unlock the focus
	FocusUnlock:		BOOL;
	FocusUnlocked:		BOOL;
	MQTTTimer : 		TON := (PT:=T#5S);
	//getlastposition:	BOOL := TRUE;
	FocusAxisEvent:		FB_EventLog;
	CalibrationEvent:	FB_EventLog;
	HomingMode: 		MC_HOMINGMODE := 		MC_DefaultHoming;
	SetPosition:		MC_SetPosition;
END_VAR

VAR CONSTANT
	// reference position for homing
	homing_position:		LREAL := 92.8936; // 106.5936 - 13.7000
	tolerance:				LREAL := 0.005;
END_VAR
VAR PERSISTENT
	last_position:		LREAL := -1.0;
END_VAR

(*
Focus Control Unit
spindle gear: 5mm
brake: 86 61103H00 Var. 0005 Index C; 24VDC geglattet 0,25 A P1672/R7
motor: Faulhaber ; Schönaich ; 3557K024CR; 454  431 ; Made in germany ==> 5300 rpm
gear: Faulhaber ; MINIMOTOR SA ; swiss made ; 38/1S  43:1 ; 033896  503
Focus is locked by default
70,8W; 0,100A no load current; 2,0 Terminal resistance; 1,950A max Current 
*)
position := LIMIT(5.0, position, 95.0);

GVL_Telescope.focus_unlock := FocusUnlock OR enable;

// wait until the focus is unlocked for n milliseconds
FocusDelay(IN := GVL_Telescope.focus_unlock, PT := T#500MS, Q => FocusUnlocked);
// wait for brake until we are at rest
BrakeDelay(IN := NOT FocusAxis.Busy AND FocusAxis.StandStill, PT := T#4000MS);

// if we are on automatic mode then position the focus
IF Pendantcontrol.telescope_mode = E_TelescopeMode.automatic AND NOT FocusUnlock THEN
	IF FocusAxis.Calibrated THEN
		IF ABS(position - actual_position) > tolerance THEN
			IF FocusAxis.Ready THEN
				MoveAxis := TRUE;
			ELSE
				Enable := TRUE;
			END_IF
		END_IF
		// disable the drive and lock the brake, if we stand for more than n seconds
		IF BrakeDelay.Q THEN
			Enable := FALSE;
		END_IF
		// store actual position, if we are calibrated and locked
		IF NOT GVL_Telescope.focus_unlock THEN
			last_position := actual_position;
		END_IF
	ELSE // not calibrated
		IF FocusAxis.Ready THEN
			HomeAxis := TRUE;
		END_IF
	END_IF
END_IF

IF HomeAxis THEN
	IF last_position > 0.0 THEN
		HomingMode := MC_ForceCalibration; // MC_Direct
		position := last_position;
		SetPosition.Execute := TRUE;
	ELSE
		HomingMode := MC_DefaultHoming;
		position := homing_position;
		SetPosition.Execute := FALSE;
	END_IF
ELSE
	SetPosition.Execute := FALSE;	
END_IF

// deactivate limit switches on homing
MC_SetAcceptBlockedDriveSignal(
	Axis := GVL_Telescope.FocusAxisRef, 
	Enable := HomeAxis);
SetPosition(
	Axis := GVL_Telescope.FocusAxisRef, 
	Position := last_position);
	
	
FocusAxis(	
	Enable := 			FocusUnlocked,
	Reset := 			reset,
	MoveAxis := 		MoveAxis AND FocusUnlocked,
	HomeAxis :=			HomeAxis AND FocusUnlocked,
	HomingMode :=		HomingMode,
	Position := 		position,
	Velocity :=			1.0,
	Enable_Positive := 	NOT GVL_Telescope.focus_limit_far OR HomeAxis,
	Enable_Negative := 	NOT GVL_Telescope.focus_limit_near,
	Jog_Forward :=		outward AND FocusUnlocked,
	Jog_Backwards := 	inward AND FocusUnlocked,
	bCalibrationCam :=  GVL_Telescope.focus_limit_far,
	ActualPosition => 	actual_position,
	Error =>			error,
	ErrorID =>			ErrorID,
	AxisRef :=			GVL_Telescope.FocusAxisRef);	

IF FocusAxis.MoveDone THEN
	MoveAxis := FALSE;
END_IF

IF FocusAxis.HomeDone THEN
	HomeAxis := FALSE;
	Enable := FALSE;
	last_position := position;
END_IF
	
IF FocusAxis.ResetDone THEN
	reset := FALSE;
END_IF

IF FocusAxis.Calibrated OR Error THEN
	HomeAxis := FALSE;
END_IF

IF Error THEN
	last_position := -1.0;
	//FocusAxis.Calibrated := FALSE;
	Calibrated := FALSE;
END_IF

Calibrated := FocusAxis.Calibrated;

Ready := FocusAxis.Ready AND FocusAxis.StandStill OR NOT GVL_Telescope.focus_unlock;

MQTTTimer(IN:=TRUE);
IF MQTTTimer.Q THEN // publish new payload every second
	MQTTTimer(IN:=FALSE);
	MAIN.MQTTClient.Publish('telescope', 'dome', 'FocusPosition', LREAL_TO_FMTSTR(actual_position, 5, TRUE));
	MAIN.MQTTClient.Publish('telescope', 'dome', 'FocusCalibrated', BOOL_TO_STRING(Calibrated));	
	MAIN.MQTTClient.Publish('telescope', 'dome', 'FocusReady', BOOL_TO_STRING(Ready));	
END_IF

FocusAxisEvent(	
	Trigger := 		FocusAxis.Error, 
	Level := 		ADSLOG_MSGTYPE_ERROR,
	FormatString :=	'Focus Axis Error: %s',
	OnMessage := 	NCError_TO_STRING(ErrorID),
	OffMEssage := 	'OK',
	OffLevel := 	ADSLOG_MSGTYPE_HINT);

CalibrationEvent(
	Trigger :=	Calibrated,
	Level :=	ADSLOG_MSGTYPE_HINT,
	OnMessage := 'Focus is calibrated.'
	);

END_PROGRAM

// ---- POUs/PendantControl.TcPOU
PROGRAM PendantControl
VAR
	// program selection of the pendant control
	Selection:	UINT;
	// error on the pendant control
	Error:		BOOL;
	// manual switch
	manual:		BOOL;
	//enable button
	enable:		BOOL;
	//reset button
	reset:		BOOL;
	// up button
	up:			BOOL;
	// down button
	down:		BOOL;
	// left button
	left:		BOOL;
	// right button
	right:		BOOL;
	lamp_left:		BOOL;
	lamp_right:		BOOL;
	lamp_up:		BOOL;
	lamp_down:		BOOL;
	lamp_error:		BOOL;
	horn:			BOOL;
	FocusEnable: 		FB_ButtonEnable;
	DerotatorEnable:	FB_ButtonEnable;
	ElevationEnable: 	FB_ButtonEnable;
	AzimuthEnable: 		FB_ButtonEnable;
	TelescopeControlEnable: 	FB_ButtonEnable;
	HydraulicsEnable: 	FB_ButtonEnable;
	TrackingEnable:			FB_ButtonEnable;
	ResetDelay:	TON;
	TwinCATRestart: TC_Restart;
	up_trigger:	R_TRIG;
	down_trigger:	R_TRIG;	
	// manual or automatic operation of the telescope
	telescope_mode : E_TelescopeMode;	
END_VAR

(* 
This program is responsible for the manual control of the telescope.
all movable parts can be controlled from here. This is mainly for testing and
maintenance.
WARNING! Some of the safety routines are disabled, when operating the telescope manually.
*)
// calculate the value of the selector
Selection := 1*BOOL_TO_UINT(GVL_pendant_control.BCD1) + 
			 2*BOOL_TO_UINT(GVL_pendant_control.BCD2) + 
			 4*BOOL_TO_UINT(GVL_pendant_control.BCD4) +
			 8*BOOL_TO_UINT(GVL_pendant_control.BCD8);

// detect disconnection of the manual controls (should also trigger emergency stop).			 
Error := (Selection = 0);

// disable all the lamps
lamp_left := FALSE;
lamp_right := FALSE;
lamp_up := FALSE;
lamp_down := FALSE;
horn := FALSE;

// clooect the state of all buttons
manual := GVL_pendant_control.key_switch;
enable := GVL_pendant_control.start_switch;
reset := GVL_pendant_control.reset_switch;
up := GVL_pendant_control.direction_up;
down := GVL_pendant_control.direction_down;
left := GVL_pendant_control.direction_left;
right := GVL_pendant_control.direction_right;

up_trigger(CLK := up);
down_trigger(CLK := down);
//R_Enable(CLK := enable);
// the error lamp is the same as the error lamp of the main panel
lamp_error := GVL_Main.lamp_error;
CoverControl.active_cover := 0;


// determine the operation of the telescope based on the switch set
IF manual THEN
	telescope_mode := E_TelescopeMode.manual;
ELSE
	telescope_mode := E_TelescopeMode.automatic;
END_IF

// enable only the selected item and connect lamps and buttons accordingly
CASE Selection OF
	1:	// reserved for Cover1 control
		lamp_up := GVL_Telescope.cover1_open;
		lamp_down := GVL_Telescope.cover1_closed;
		IF manual THEN
			//CoverEnable(SET := enable, Q := CoverControl.enable);
			//CoverControl.active_cover := 1;
			//CoverControl.reset := reset;
			GVL_Telescope.open_cover1 := up AND GVL_Telescope.cover1_open;
			GVL_Telescope.close_cover1 := down AND GVL_Telescope.cover1_closed;
			lamp_error := CoverControl.Cover1_Error;	
		ELSE
			IF down THEN 
				CoverControl.close := TRUE;
			END_IF
			IF up THEN
				CoverControl.open := TRUE;
			END_IF		
		END_IF

	2: // Cover2 control
		lamp_up := GVL_Telescope.cover2_open;
		lamp_down := GVL_Telescope.cover2_closed;
		IF manual THEN
			//CoverEnable(SET := enable, Q := CoverControl.enable);
			//CoverControl.active_cover := 2;
			GVL_Telescope.open_cover2 := up AND GVL_Telescope.cover2_open;
			GVL_Telescope.close_cover2 := down AND GVL_Telescope.cover2_closed;
			lamp_error := CoverControl.Cover2_Error;
		ELSE
			IF down THEN 
				CoverControl.close := TRUE;
			END_IF
			IF up THEN
				CoverControl.open := TRUE;
			END_IF		
		END_IF
 	
	3:  // Cover3 control
		lamp_up := GVL_Telescope.cover3_open;
		lamp_down := GVL_Telescope.cover3_closed;
		IF manual THEN
			//CoverEnable(SET := enable, Q := CoverControl.enable);
			//CoverControl.active_cover := 3;
			GVL_Telescope.open_cover3 := up AND GVL_Telescope.cover3_open;
			GVL_Telescope.close_cover3 := down AND GVL_Telescope.cover3_closed;
			//CoverControl.reset := reset;
			lamp_error := CoverControl.Cover3_Error;
		ELSE
			IF down THEN 
				CoverControl.close := TRUE;
			END_IF
			IF up THEN
				CoverControl.open := TRUE;
			END_IF		
		END_IF
		
	4:	// Nasmyth / mirror M3 control
		
	5:	// Focus Control
		lamp_up := FocusControl.Ready AND NOT GVL_Telescope.focus_limit_far;
		lamp_down := FocusControl.Ready AND NOT GVL_Telescope.focus_limit_near;
		IF manual THEN
			FocusEnable(SET := enable, Q := FocusControl.enable);
			FocusControl.outward := up;
			FocusControl.inward := down;
			Focuscontrol.reset := reset;
			lamp_error := FocusControl.error;
		END_IF
							
	6:	// Derotator control
		lamp_left := DerotatorControl.Ready AND NOT GVL_Telescope.Derotator_inputs.1;
		lamp_right :=DerotatorControl.Ready AND NOT GVL_Telescope.Derotator_inputs.0;
		IF manual THEN
			DerotatorEnable(SET := enable, Q := DerotatorControl.enable);
			DerotatorControl.left := left AND NOT GVL_Telescope.Derotator_inputs.1;
			DerotatorControl.right := right AND NOT GVL_Telescope.Derotator_inputs.0;
			DerotatorControl.reset := reset;
			lamp_error := DerotatorControl.Error;
		END_IF
							
	7:	// Elevation Control
		
		ElevationControl.up := up AND GVL_Telescope.Elevation_inputs.0;
		ElevationControl.down := down AND GVL_Telescope.Elevation_inputs.1;
		IF manual THEN
			ElevationEnable(
				SET := enable, 
				Q := ElevationControl.enable);	
		END_IF
		ElevationControl.reset := reset;
		lamp_up := GVL_Telescope.Elevation_inputs.0;
		lamp_down := GVL_Telescope.Elevation_inputs.1;
		lamp_error := ElevationControl.error;
		
	8:	// Azimuth Control
		lamp_left := GVL_Telescope.Azimuth_inputs.0; // NOT GVL_Telescope.azimut_limit_switch;
		lamp_right := GVL_Telescope.Azimuth_inputs.1; // NOT GVL_Telescope.azimut_limit_switch;
		AzimuthElevationControl.left := left AND GVL_Telescope.Azimuth_inputs.0;
		AzimuthElevationControl.right := right AND GVL_Telescope.Azimuth_inputs.1;
		AzimuthElevationControl.reset := reset;
		IF manual THEN
			AzimuthEnable(
				SET := enable, 
				Q := AzimuthElevationControl.enable);
			lamp_error := AzimuthElevationControl.error;
		END_IF
		
	9: 	// Dome control
		
	10:	// FilterWheel control
		
	11: lamp_up := ElevationControl.elevation_torque > 0.0;
		lamp_down := ElevationControl.elevation_torque < 0.0;
		
	12:	// manual Telescope Control
		IF manual THEN
			lamp_up := TelescopeControl.power;
			lamp_down := TelescopeControl.power;
			lamp_left := TelescopeControl.power;
			lamp_right := TelescopeControl.power;
	
			TelescopeControl.gohome := down;
			TelescopeControl.park := up;
			TelescopeControl.goto := right;
			TrackingEnable(SET := enable, 
							RESET := reset, 
							Q := TelescopeControl.track);
			TelescopeControl.reset := reset;
			Telescopecontrol.stop := left;	
			lamp_error := Telescopecontrol.error;
		END_IF
		
	13: // Telescope Control
		TelescopeControlEnable(
			SET := enable, 
			Q := TelescopeControl.power);
		TelescopeControl.reset := reset;
		IF manual THEN
			lamp_up := GVL_Telescope.Elevation_inputs.0;
			lamp_down := GVL_Telescope.Elevation_inputs.1;
			lamp_left := GVL_Telescope.Azimuth_inputs.0;
			lamp_right := GVL_Telescope.Azimuth_inputs.1;
			ElevationControl.up := up AND GVL_Telescope.Elevation_inputs.0;
			ElevationControl.down := down AND GVL_Telescope.Elevation_inputs.1;
			AzimuthElevationControl.left := left AND GVL_Telescope.Azimuth_inputs.0;
			AzimuthElevationControl.right := right AND GVL_Telescope.Azimuth_inputs.1;
			TelescopeControl.rightascension := TelescopeControl.rightascension_calc;
			TelescopeControl.declination := TelescopeControl.declination_calc;
		ELSE
			lamp_up := ElevationControl.enable;
			lamp_down := ElevationControl.enable;
			lamp_left := AzimuthElevationControl.enable;
			lamp_right := AzimuthElevationControl.enable;
			IF up THEN 
				Telescopecontrol.elevation_offset := Telescopecontrol.elevation_offset + 10.0/3600.0; 
			ELSIF down THEN 
				Telescopecontrol.elevation_offset := Telescopecontrol.elevation_offset - 10.0/3600.0; 
			END_IF;
			IF left THEN 
				Telescopecontrol.azimuth_offset := Telescopecontrol.azimuth_offset - 10.0/3600.0; 
			ELSIF right THEN 
				Telescopecontrol.azimuth_offset := Telescopecontrol.azimuth_offset + 10.0/3600.0; 
			END_IF;
		END_IF
		ResetDelay(IN := reset, PT := T#3S);
		// wait for suction pump to stop
		TwinCATRestart(NETID := '', RESTART := ResetDelay.Q AND NOT HydraulicsControl.suction_running, TMOUT := T#60S);
	
	14: horn := manual;
		lamp_up := manual;
		lamp_down := manual;
		lamp_left := manual;
		lamp_right := manual;
	
	15:	// Hydraulics control
		lamp_up := HydraulicsControl.oil_pressure_OK AND Hydraulicscontrol.brake_closed;
		lamp_down := HydraulicsControl.oil_pressure_OK AND Hydraulicscontrol.brake_open;
		lamp_left := HydraulicsControl.pump_running;
		lamp_right := HydraulicsControl.suction_running;
		IF manual THEN
			HydraulicsEnable(
				SET := enable, 
				Q := Hydraulicscontrol.enable);
			Hydraulicscontrol.reset := reset;
			
			IF up THEN
				Hydraulicscontrol.open_brake();
			END_IF
			IF down THEN
				Hydraulicscontrol.close_brake();
			END_IF
			Hydraulicscontrol.suction_manual := right;
			Hydraulicscontrol.pump_manual_stop := left;
			lamp_error := HydraulicsControl.error;
		END_IF
END_CASE

// set all the lamps
GVL_pendant_control.lamp_left := lamp_left;
GVL_pendant_control.lamp_right := lamp_right;
GVL_pendant_control.lamp_up := lamp_up;
GVL_pendant_control.lamp_down := lamp_down;
GVL_pendant_control.lamp_error := lamp_error;

END_PROGRAM

// ---- POUs/TelescopeControl.TcPOU
PROGRAM TelescopeControl
VAR_INPUT
(*
TCS interface section
see https://gitlab.aip.de/bmk10k/telescope_firmware/snippets/5
*)
	
	// boolean, true: Power on, false: power off
	power: 		BOOL;
	// boolean, true: go to home position, unset track/goto if active
	gohome: 	BOOL;
	// boolean, true: go into park position, ready to stow telescope, unset track/goto
	park: 		BOOL;
	// boolean, TRUE: MOVE telescope TO last ra/de AND start tracking. Set 'goto' TO FALSE, IF TRUE. FALSE: Stop tracking as soon as possible
	track: 		BOOL;
	// boolean, TRUE: MOVE telescope TO tau/de AND stop there. Set track TO FALSE, IF TRUE. FALSE: no effect.)
	goto:		BOOL;	
	// move the telescope to a given az-alt position
	slew:		BOOL;
	// boolean, TRUE: Stop motion OF telescope immediately, set goto AND track TO FALSE. FALSE: Allow motion OF telescope again via track/goto).
	stop:		BOOL;	
	// initiates reset on all axis
	reset:		BOOL;
	// automatic tracking after goto
	autotrack:	BOOL := TRUE;
	// apparent right ascension, degrees, double
	rightascension:		LREAL := (4.0 + 35.0/60.0 + 54.09/3600.0) *15.0;	
	// apparent declination, degrees, double
	declination: 		LREAL := 16.0 + 30.0/60.0 + 25.4/3600.0;
	// desired elevation of the telescope pointing 
	elevation:	LREAL := 45.0;
	// desired azimut of the telescope pointing 
	azimuth:	LREAL := 320.0;
	// absolute offset for elevation
	elevation_offset:	LREAL := 0.0;
	// absolute offset for azimuth
	azimuth_offset : 	LREAL := 0.0;
	// absolute offset for time
	time_offset: 		LREAL := 0.0;
	// offset for the de-rotator
	derotator_offset:	LREAL := 0.0;
END_VAR
VAR
	// actual command from the TCS
	TCS_command: 	E_TCSCommand;
	// current Julian Date calculated from system time
	jd:				LREAL;
	// image derotation
	derotation_calc:	LREAL;
	// local siderial time calculated from Julian date
	lst:			LREAL;
	// elevation calulated when ra and dec are set by TCS
	elevation_calc:	LREAL; 
	// azimuth calulated when ra and dec are set by TCS
	azimuth_calc:	LREAL;
	// right ascension calulated when azimuth and elevation are set by TCS
	rightascension_calc:	LREAL;
	// declination calulated when azimuth and elevation are set by TCS
	declination_calc:		LREAL;
	// hour angle
	Hourangle_calc: LREAL;
	// precise astronomical	time
	fbTime: FB_AstroClock;
	
	eq2hor:		FB_EQ2HOR;
	hor2eq:		FB_HOR2EQ;
	
	// triggers power-failure event
	powerfailure: 	BOOL;
	// triggers power warning
	poweronwarning:	TP;
	// power on timeout
	power_timeout:	TON;
	// tracking delay
	tracking_delay:	TON;
	// telescope is parked
	isparked:		BOOL;
	TCSpowerEvent,
	TCSgohomeEvent,
	TCSparkEvent,
	TCSgotoEvent,
	TCStrackEvent,
	TCSstopEvent,
	AltitudeEvent,
	TCSreadyEvent: FB_Eventlog;
	MQTTTimer : TON := (PT:=T#5S);
	// rotational velocity of the derotator
	DerotatorVelocity: LREAL;
	// rotational velocity of the elevation
	ElevationVelocity: LREAL;
	// rotational velocity of the elevation
	AzimuthVelocity: LREAL;
	// sign of derotation
	derotatation_sign: LREAL := 1.0;
	StatusWord, LastStatus:	UDINT;
END_VAR
VAR_OUTPUT
	//		TRUE, IF telescope can be operated
	ready:		BOOL; 
	// indicates an error on one of the components
	error:		BOOL;	
	//error id of axis
	errorid:	UDINT;	
	//TRUE, IF telescope is in fast-MOVE phase (includes pole-swap)
	sliding:	BOOL;	
	//TRUE, IF telescope is on tracking position AND currently tracking.
	tracking:	BOOL;	
	//TRUE, IF telescope is AT rest.
	stopped:	BOOL;	
	// true position of the elevation
	elevation_current:	LREAL;
	// true position of the azimuth
	azimuth_current:	LREAL;
	// true position of the de-rotator
	derotator_current:	LREAL;
	//	(time in sec. to reach the goto/track position)
	slewtime:			LREAL; 
	// True: telescope is calibrated
	homed:				BOOL;
	// telescope does not accept further commands
	busy:				BOOL;
END_VAR
VAR CONSTANT
// STELLA1
	// telescope site longitude, source: Google 
	longitude: 		LREAL := -16.50926; //13.101867;
	// telescope site latitude, source: Google
	latitude: 		LREAL := 28.30120; //52.404940;
	// telescope site height above sea level: estimated
	altitude: 		LREAL := 2390.0;
	elevation_park: LREAL := 60.0;
	azimuth_park: 	LREAL := 359.999;
	derotator_park: LREAL := 229.85;

	elevation_home: LREAL := 55.0;
	azimuth_home: 	LREAL := 180.0;
END_VAR
VAR PERSISTENT
	// azimuth axis offset/misalignment north-south
	AN_E:	LREAL;
	// azimuth axis offset/misalignment east-west
	AE_E:	LREAL;
	// gravitational flexure correction at the horizon
	TF:		LREAL;
	// collimation error of the electromagnetic axis
	BNP:	LREAL;
	// azimuth axis offset/misalignment north-south
	AN_A:	LREAL;
	// azimuth axis offset/misalignment east-west,
	AE_A:	LREAL;
	// Non-perpendicularity between the mount azimuth and elevation axes
	NPAE:	LREAL;
END_VAR

TelescopeAuxiliary();

// get the system time
fbTime();
jd := DateTime2JD(fbTime.time_RTCEX2);
lst := CT2LST(longitude, jd);
// set reset state either by hardware (key pressed) or by software (set by e.g. tcs)
IF GVL_Main.reset_switch THEN
	reset := TRUE;
END_IF


IF ElevationControl.error THEN
	errorid := ElevationControl.ErrorID;
	ElevationControl.reset := reset;
ELSIF AzimuthElevationControl.error THEN
	errorid := AzimuthElevationControl.ErrorID;
	AzimuthElevationControl.Reset := reset;
ELSIF Focuscontrol.Error THEN
	errorid := Focuscontrol.ErrorID;
	FocusControl.reset := reset;
ELSIF DerotatorControl.Error THEN
	errorid := DerotatorControl.ErrorID;
	DerotatorControl.reset := reset;
END_IF

error := ElevationControl.error OR 
		 AzimuthElevationControl.error OR
		 Focuscontrol.Error OR
		 DerotatorControl.Error;

slewtime := MAX(MAX(ElevationControl.slewtime, AzimuthElevationControl.slewtime), DerotatorControl.slewtime);
			
IF error THEN
	gohome := 	FALSE;
	track := 	FALSE;
	goto := 	FALSE;
	slew := 	FALSE;
ELSE
	errorid := 0;
END_IF

IF ElevationControl.error THEN
	ElevationControl.enable := FALSE;
	AzimuthElevationControl.enable := FALSE;
	HydraulicsControl.close_brake();
END_IF

eq2hor(
	ra := rightascension,
	dec := declination,
	lon := longitude,
	lat := latitude,
	JD := jd + time_offset,
	alt => elevation_calc,
	az => azimuth_calc,
	ha => hourangle_calc);

// apply pointing model
elevation_calc := elevation_calc + PointingModelElevation(azimuth_calc, elevation_calc, elevation_offset, AN_E, AE_E, TF);
azimuth_calc := azimuth_calc + PointingModelAzimuth(azimuth_calc, elevation_calc, azimuth_offset, BNP, AN_A, AE_A, NPAE);
// calculate derotator position 
derotation_calc := F_DerotatorPosition2(azimuth_calc, elevation_calc, declination_calc, latitude, derotatation_sign)  + derotator_offset;
// calculate velocities
DerotatorVelocity := F_Derotatorvelocity(elevation_calc, azimuth_calc, latitude);
ElevationVelocity := F_Elevationvelocity(azimuth_calc, latitude);
AzimuthVelocity := F_Azimuthvelocity(elevation_calc, azimuth_calc, latitude);

IF (azimuth_calc > 310.0 AND AzimuthVelocity > 0.0) OR (azimuth_calc > 440.0) THEN
	azimuth_calc := azimuth_calc - 360.0;
ELSIF (azimuth_calc < 80.0 AND AzimuthVelocity < 0.0) OR (azimuth_calc < -50.0) THEN
	azimuth_calc := azimuth_calc + 360.0;
END_IF

IF (derotation_calc > 290.0 AND DerotatorVelocity > 0.0) OR (derotation_calc > 380.0) THEN
	derotation_calc := derotation_calc - 360.0;
ELSIF (derotation_calc < 20.0 AND DerotatorVelocity < 0.0) OR (derotation_calc < -70.0) THEN
	derotation_calc := derotation_calc + 360.0;
END_IF
// get current coordinates	
azimuth_current := AzimuthElevationControl.act_position;
elevation_current := ElevationControl.actual_position;
derotator_current := DerotatorControl.actual_position;

// calculate equatorial coordinates
hor2eq(alt := elevation_current - PointingModelElevation(azimuth_calc, elevation_calc, elevation_offset, AN_E, AE_E, TF), 
		az := azimuth_current - PointingModelAzimuth(azimuth_calc, elevation_calc, azimuth_offset, BNP, AN_A, AE_A, NPAE),
		jd := jd,
		lat := latitude,
		lon := longitude,
		altitude := altitude,
		ra => rightascension_calc,
		dec => declination_calc);		
	
poweronwarning(IN := power OR (NOT ElevationControl.enable AND HydraulicsControl.brake_open), PT := T#250MS);

power_timeout(IN := TCS_command = E_TCSCommand.no_command AND NOT isparked, PT := T#12H);
IF power_timeout.Q AND NOT isparked THEN
	park := TRUE;
END_IF
		
// set TCS_command according to state variables ordered by precedence
IF power THEN
	TCS_command := E_TCSCommand.poweron;
ELSIF stop THEN
	TCS_command := E_TCSCommand.stop;
	goto := FALSE;
	track := FALSE;
	slew := FALSE;
	gohome := FALSE;
	park := FALSE;
ELSIF park THEN
	TCS_command := E_TCSCommand.park;
	goto := FALSE;
	track := FALSE;
	slew := FALSE;
ELSIF gohome THEN
	goto := FALSE;
	track := FALSE;
	slew := FALSE;
	IF ready AND NOT busy THEN
		TCS_command := E_TCSCommand.gohome;
	END_IF
ELSIF goto THEN
	track := FALSE;
	slew := FALSE;
	IF ready AND NOT busy THEN
		TCS_command := E_TCSCommand.goto;
	END_IF
ELSIF slew THEN
	goto := FALSE;
	track := FALSE;
	IF ready AND NOT busy THEN
		TCS_command := E_TCSCommand.slew;
	END_IF
ELSIF track THEN
	goto := FALSE;
	slew := FALSE;
	IF ready AND NOT busy THEN
		TCS_command := E_TCSCommand.track;
	END_IF
ELSE
	TCS_command := E_TCSCommand.no_command;
	ElevationControl.MoveAxis := FALSE;
	AzimuthElevationControl.MoveAxis := FALSE;
	DerotatorControl.MoveAxis := FALSE;
	ElevationControl.Tracking := FALSE;
	AzimuthElevationControl.Tracking := FALSE;
	DerotatorControl.Tracking := FALSE;
END_IF

IF TCS_command = E_TCSCommand.poweron THEN
	poweron();
ELSIF TCS_command = E_TCSCommand.stop THEN
	stoptelescope();
ELSIF TCS_command = E_TCSCommand.park THEN
	parktelescope();
ELSIF TCS_command = E_TCSCommand.gohome THEN
	hometelescope();
ELSIF TCS_command = E_TCSCommand.goto THEN
	gototelescope();
ELSIF TCS_command = E_TCSCommand.slew THEN
	slewtelescope();
ELSIF TCS_command = E_TCSCommand.track THEN
	tracktelescope();
END_IF
 
sliding := NOT tracking AND (ElevationControl.ElevationAxis.InMotion OR ElevationControl.ElevationAxis.InRamp OR
			AzimuthElevationControl.AzimuthAxis.InMotion OR AzimuthElevationControl.AzimuthAxis.InRamp OR
			DerotatorControl.DerotatorAxis.InMotion OR DerotatorControl.DerotatorAxis.InRamp);

// signal must be stable for 3000MS			
tracking_delay(in := ElevationControl.ElevationAxis.isTracking AND 
			AzimuthElevationControl.AzimuthAxis.isTracking AND
			DerotatorControl.DerotatorAxis.isTracking,PT :=T#5500MS, Q => tracking);
			
stopped :=  (NOT ElevationControl.enable OR ElevationControl.ElevationAxis.StandStill) AND 
			(NOT AzimuthElevationControl.Enable OR AzimuthElevationControl.AzimuthAxis.StandStill) AND
			(NOT DerotatorControl.enable OR DerotatorControl.DerotatorAxis.StandStill);
			
homed := ElevationControl.Calibrated AND
			AzimuthElevationControl.calibrated AND
			FocusControl.Calibrated AND
			DerotatorControl.Calibrated;
			
ready := homed AND 
	CoverControl.isopen AND 
	ElevationControl.enable AND
	AzimuthElevationControl.enable AND
	DerotatorControl.enable AND HydraulicsControl.brake_open AND 
    NOT error;

busy := ElevationControl.ElevationAxis.Busy OR
		AzimuthElevationControl.AzimuthAxis.Busy OR
		DerotatorControl.DerotatorAxis.Busy OR
		FocusControl.FocusAxis.Busy;
	
IF NOT error THEN
	reset := FALSE;
END_IF

IF SafetyHandling.Emergency_stop THEN
	ElevationControl.enable := FALSE;
	AzimuthElevationControl.enable := FALSE;
	DerotatorControl.enable := FALSE;
END_IF
IF sliding OR track OR tracking THEN
	MQTTTimer.PT := T#1000MS;
ELSE
	MQTTTimer.PT := T#5000MS;
END_IF
MQTTTimer(IN:=TRUE);
IF MQTTTimer.Q THEN // publish new payload every second
	MQTTTimer(IN:=FALSE);

	MAIN.MQTTClient.Publish('telescope', 'dome', 'JulianDate', LREAL_TO_STRING(jd));
	MAIN.MQTTClient.Publish('telescope', 'dome', 'LocalSiderialTime', LREAL_TO_STRING(lst));
	MAIN.MQTTClient.Publish('telescope', 'dome', 'Azimuth', LREAL_TO_STRING(azimuth_current));
	MAIN.MQTTClient.Publish('telescope', 'dome', 'Elevation', LREAL_TO_STRING(elevation_current));
	MAIN.MQTTClient.Publish('telescope', 'dome', 'Derotator', LREAL_TO_STRING(derotator_current));
	MAIN.MQTTClient.Publish('telescope', 'dome', 'HourAngle', LREAL_TO_STRING(hourangle_calc));
	MAIN.MQTTClient.Publish('telescope', 'dome', 'RightAscension', LREAL_TO_STRING(rightascension_calc));
	MAIN.MQTTClient.Publish('telescope', 'dome', 'Declination', LREAL_TO_STRING(declination_calc));
	MAIN.MQTTClient.Publish('telescope', 'dome', 'azimuth_offset', LREAL_TO_STRING(azimuth_offset));
	MAIN.MQTTClient.Publish('telescope', 'dome', 'elevation_offset', LREAL_TO_STRING(elevation_offset));
	MAIN.MQTTClient.Publish('telescope', 'dome', 'derotator_torque', LREAL_TO_STRING(DerotatorControl.derotator_torque));
	MAIN.MQTTClient.Publish('telescope', 'dome', 'elevation_torque', LREAL_TO_STRING(ElevationControl.elevation_torque));
	MAIN.MQTTClient.Publish('telescope', 'dome', 'azimuth_torque', LREAL_TO_STRING(AzimuthElevationControl.azimuth_torque));
	
	MAIN.MQTTClient.Publish('telescope', 'dome', 'errorid',		UDINT_TO_STRING(errorid));
	MAIN.MQTTClient.Publish('telescope', 'dome', 'error',		BOOL_TO_STRING(error));
	MAIN.MQTTClient.Publish('telescope', 'dome', 'ready',		BOOL_TO_STRING(ready));
	MAIN.MQTTClient.Publish('telescope', 'dome', 'busy',		BOOL_TO_STRING(busy));
	MAIN.MQTTClient.Publish('telescope', 'dome', 'sliding',		BOOL_TO_STRING(sliding));
	MAIN.MQTTClient.Publish('telescope', 'dome', 'tracking', 	BOOL_TO_STRING(tracking));
	MAIN.MQTTClient.Publish('telescope', 'dome', 'stopped',		BOOL_TO_STRING(stopped));
	MAIN.MQTTClient.Publish('telescope', 'dome', 'homed',		BOOL_TO_STRING(homed));
END_IF

StatusWord.0 := error;
StatusWord.1 := ready;
StatusWord.2 := sliding;
StatusWord.3 := tracking;
StatusWord.4 := stopped;
StatusWord.5 := homed;
StatusWord.6 := power;
StatusWord.7 := park;
StatusWord.8 := gohome;
StatusWord.9 := track;
StatusWord.10 := goto;
StatusWord.11 := slew;
StatusWord.12 := stop;
StatusWord.13 := busy;

IF StatusWord<>LastStatus THEN // publish new payload every second
	LastStatus := StatusWord;
	MAIN.MQTTClient.Publish('telescope', 'dome', 'error',		BOOL_TO_STRING(error));
	MAIN.MQTTClient.Publish('telescope', 'dome', 'ready',		BOOL_TO_STRING(ready));
	MAIN.MQTTClient.Publish('telescope', 'dome', 'sliding',		BOOL_TO_STRING(sliding));
	MAIN.MQTTClient.Publish('telescope', 'dome', 'tracking', 	BOOL_TO_STRING(tracking));
	MAIN.MQTTClient.Publish('telescope', 'dome', 'stopped',		BOOL_TO_STRING(stopped));
	MAIN.MQTTClient.Publish('telescope', 'dome', 'homed',		BOOL_TO_STRING(homed));
	MAIN.MQTTClient.Publish('telescope', 'dome', 'power',		BOOL_TO_STRING(power));
	MAIN.MQTTClient.Publish('telescope', 'dome', 'park',		BOOL_TO_STRING(park));
	MAIN.MQTTClient.Publish('telescope', 'dome', 'gohome',		BOOL_TO_STRING(gohome));
	MAIN.MQTTClient.Publish('telescope', 'dome', 'track',		BOOL_TO_STRING(track));
	MAIN.MQTTClient.Publish('telescope', 'dome', 'goto',		BOOL_TO_STRING(goto));
	MAIN.MQTTClient.Publish('telescope', 'dome', 'slew',		BOOL_TO_STRING(slew));
	MAIN.MQTTClient.Publish('telescope', 'dome', 'stop',		BOOL_TO_STRING(stop));
	MAIN.MQTTClient.Publish('telescope', 'dome', 'busy',		BOOL_TO_STRING(busy));
END_IF


(* Event function blocks start here. *)
TCSpowerEvent(	Trigger := powerfailure, 
				Level := ADSLOG_MSGTYPE_ERROR,
				FormatString := 'power %s',
				OnMessage := 'Failure',
				OffMessage := 'OK');

TCSgohomeEvent(	Trigger := gohome, 
				Level := ADSLOG_MSGTYPE_HINT,
				FormatString := 'GOHOME %s',
				OnMessage := 'commencing',
				OffMEssage := 'completed');
TCSparkEvent(	Trigger := park, 
				Level := ADSLOG_MSGTYPE_HINT,
				FormatString := 'PARK %s',
				OnMessage := 'commencing',
				OffMEssage := 'completed');
TCSgotoEvent(	Trigger := goto, 
				Level := ADSLOG_MSGTYPE_HINT,
				FormatString := 'GOTO %s',
				OnMessage := 'commencing',
				OffMEssage := 'completed');
TCStrackEvent(	Trigger := track, 
				Level := ADSLOG_MSGTYPE_HINT,
				FormatString := 'TRACK %s',
				OnMessage := 'commencing',
				OffMEssage := 'completed');
TCSstopEvent(	Trigger := stop, 
				Level := ADSLOG_MSGTYPE_WARN,
				FormatString := 'STOP %s',
				OnMessage := 'commencing',
				OffMEssage := 'completed',
				OffLevel := ADSLOG_MSGTYPE_HINT);
AltitudeEvent(	Trigger := power AND elevation_calc<0.0, 
				Level := ADSLOG_MSGTYPE_WARN,
				FormatString := '%s',
				OnMessage := 'Target below horizon',
				OffMEssage := '');
TCSreadyEvent(	Trigger := power AND ready, 
				Level := ADSLOG_MSGTYPE_HINT,
				FormatString := '%s',
				OnMessage := 'STELLA1 startup finished');

METHOD gototelescope: USINT
VAR_INPUT
END_VAR
VAR
	GoToEvent:	FB_Eventlog;
	command_timeout:	TON;
END_VAR
VAR_STAT
	Stage:		USINT := 0;
	LastStage:	USINT := 101;
END_VAR
gototelescope := Stage;
command_timeout(IN := Stage < 100, PT := T#600S);
IF command_timeout.Q THEN
	error := TRUE;
	errorid := 16#10;
	goto := FALSE;
	Stage := 0;
	RETURN;
END_IF

IF elevation_calc<2.0 THEN
	error := TRUE;
	errorid := 16#15;
	goto := FALSE;
	Stage := 0;
	RETURN;
END_IF

IF reset OR error THEN
	Stage := 0;
	RETURN;
END_IF

CASE Stage OF
	0:	
		IF ready AND NOT busy THEN
			Stage := 25;
		END_IF
	25:	
		ElevationControl.position := elevation_calc;
		AzimuthElevationControl.position := azimuth_calc;
		DerotatorControl.position := derotation_calc;
		DerotatorControl.Velocity := 10.0;
		ElevationControl.velocity := 10.0;
		AzimuthElevationControl.velocity := 10.0;
		
		ElevationControl.MoveAxis := TRUE;
		AzimuthElevationControl.MoveAxis := TRUE;
		DerotatorControl.MoveAxis := TRUE;
		IF ElevationControl.ElevationAxis.Busy AND
			AzimuthElevationControl.AzimuthAxis.Busy AND
			DerotatorControl.DerotatorAxis.Busy THEN
				Stage := 50;
		END_IF
	50:
		IF NOT ElevationControl.ElevationAxis.Busy AND ElevationControl.ElevationAxis.MoveDone THEN
			ElevationControl.MoveAxis := FALSE;
		END_IF
		IF NOT AzimuthElevationControl.AzimuthAxis.Busy AND AzimuthElevationControl.AzimuthAxis.MoveDone THEN
			AzimuthElevationControl.MoveAxis := FALSE;
		END_IF
		IF NOT DerotatorControl.DerotatorAxis.Busy AND DerotatorControl.DerotatorAxis.MoveDone THEN
			DerotatorControl.MoveAxis := FALSE;
		END_IF
		IF NOT ElevationControl.MoveAxis AND 
           NOT AzimuthElevationControl.MoveAxis AND 
		   NOT DerotatorControl.MoveAxis THEN
		   Stage := 75;
		END_IF
	75:
		IF NOT sliding AND stopped THEN // all axis standstill
			Stage := 100;
		END_IF
	100:
		ElevationControl.MoveAxis := FALSE;
		AzimuthElevationControl.MoveAxis := FALSE;
		DerotatorControl.MoveAxis := FALSE;
		azimuth := azimuth_calc;
		elevation := elevation_calc;
		goto := FALSE;
		// enable automatic tracking
		track := autotrack;
		Stage := 0;
END_CASE
GoToEvent(Trigger := Stage > LastStage, FormatString := 'GoTo progress: %s', OnMessage := USINT_TO_STRING(Stage));
LastStage := Stage;
END_METHOD

METHOD hometelescope : BOOL
VAR_INPUT
END_VAR

VAR
	HomeEvent: FB_Eventlog;
	command_timeout: TON;
END_VAR
command_timeout(IN := NOT hometelescope, PT := T#600S);
IF command_timeout.Q THEN
	error := TRUE;
	errorid := 16#30;
	hometelescope :=TRUE;
END_IF

IF ready AND stopped AND NOT busy AND NOT tracking THEN
	ElevationControl.velocity := 10.0;
	ElevationControl.position := elevation_home;
	ElevationControl.MoveAxis := TRUE;
	AzimuthElevationControl.velocity := 10.0;
	AzimuthElevationControl.position := azimuth_home;
	AzimuthElevationControl.MoveAxis := TRUE;
	DerotatorControl.Velocity := 10.0;
	DerotatorControl.position := 180.0;
	DerotatorControl.MoveAxis := TRUE;	
END_IF

IF ElevationControl.ElevationAxis.MoveDone AND 
	AzimuthElevationControl.AzimuthAxis.MoveDone AND 
	DerotatorControl.DerotatorAxis.MoveDone THEN
	gohome := FALSE;
	elevation := elevation_current;
	azimuth := azimuth_current;
	hometelescope := TRUE;
ELSE
	hometelescope := FALSE;
END_IF

HomeEvent(Trigger := hometelescope, 
			Level := ADSLOG_MSGTYPE_HINT,
			FormatString := '%s',
			OnMessage := 'Telescope is homed.');
END_METHOD

METHOD parktelescope: USINT
VAR_INPUT
END_VAR
VAR
	ParkEvent:	FB_Eventlog;
	command_timeout:	TON;
END_VAR
VAR_STAT
	Stage:		USINT := 0;
	LastStage:	USINT := 101;
END_VAR
parktelescope := Stage;
command_timeout(IN := Stage < 100, PT := T#600S);
IF command_timeout.Q THEN
	error := TRUE;
	errorid := 16#20;
	Stage := 0;
END_IF
IF reset OR error THEN
	Stage := 0;
END_IF
IF isparked THEN
	Stage := 100;
END_IF
CASE Stage OF
	0: 
		gohome := 	FALSE;
		track := 	FALSE;
		goto := 	FALSE;
		slew := 	FALSE;
		Focuscontrol.position := 53.6;
		IF Error THEN // emergency park
			HydraulicsControl.close_brake();
			ElevationControl.enable := FALSE;
			AzimuthElevationControl.Enable := FALSE;
			DerotatorControl.enable := FALSE;	
			CoverControl.close := TRUE;	
			Stage := 80;
		END_IF
		Stage := 20;
	20:
		ElevationControl.position := elevation_park;
		ElevationControl.velocity := 10.0;
		ElevationControl.MoveAxis := TRUE;
		AzimuthElevationControl.position := azimuth_park;
		AzimuthElevationControl.velocity := 10;
		AzimuthElevationControl.MoveAxis := TRUE;
		DerotatorControl.position := derotator_park;
		DerotatorControl.Velocity := 10.0;
		DerotatorControl.MoveAxis := TRUE;
		IF ElevationControl.ElevationAxis.Busy AND
			AzimuthElevationControl.AzimuthAxis.Busy AND
			DerotatorControl.DerotatorAxis.Busy THEN
				Stage := 40;
		END_IF
	40:
		IF ElevationControl.ElevationAxis.MoveDone THEN
			ElevationControl.MoveAxis := FALSE;
		END_IF
		IF AzimuthElevationControl.AzimuthAxis.MoveDone THEN
			AzimuthElevationControl.MoveAxis := FALSE;
		END_IF
		IF DerotatorControl.DerotatorAxis.MoveDone THEN
			DerotatorControl.MoveAxis := FALSE;
		END_IF
		IF NOT sliding THEN // all axis standstill
			Stage := 60;
		END_IF
	60:
		IF stopped THEN 
			ElevationControl.enable := FALSE;
			AzimuthElevationControl.Enable := FALSE;
			DerotatorControl.enable := FALSE;
			Stage := 80;
		END_IF
		
		ElevationControl.MoveAxis := FALSE;
		AzimuthElevationControl.MoveAxis := FALSE;
		DerotatorControl.MoveAxis := FALSE;
	80:
		IF HydraulicsControl.brake_closed THEN
			CoverControl.close := TRUE;			
		END_IF
		IF CoverControl.isclosed THEN
			Stage := 100;
		END_IF
	100:
			isparked := TRUE;
			park := FALSE;
			parktelescope := 100;
			Stage := 0;	
END_CASE
ParkEvent(Trigger := Stage > LastStage, FormatString := 'Parking progress: %s', OnMessage := USINT_TO_STRING(Stage));
LastStage := Stage;
END_METHOD

METHOD poweron : BOOL
VAR_INPUT
END_VAR
VAR
END_VAR
IF NOT Main.brake_clearing THEN
	powerfailure := TRUE;
	TCSpowerEvent.OnMessage := 'failure: brake clearing not set';
	power := FALSE;
ELSIF error THEN
	powerfailure := TRUE;
	TCSpowerEvent.OnMessage := 'Generic error during power on occured.';
	power := FALSE;
ELSE
	powerfailure := FALSE;		
END_IF
// COVER MUST BE OPENED FOR A SUCCESSFUL WAKE & SHAKE COMMAND!
Covercontrol.open := TRUE;

// enable elevation, enable azimuth
IF MAIN.ready AND CoverControl.isopen THEN
	ElevationControl.enable := TRUE;
	AzimuthElevationControl.enable := TRUE;
	DerotatorControl.enable := TRUE;
END_IF

IF ElevationControl.Ready AND NOT ElevationControl.Calibrated THEN
	ElevationControl.HomeAxis := TRUE;
END_IF

IF AzimuthElevationControl.ready AND NOT AzimuthElevationControl.calibrated THEN
	AzimuthElevationControl.HomeAxis := TRUE;
END_IF

// enable derotator
IF ElevationControl.Ready THEN
	DerotatorControl.HomeAxis := DerotatorControl.Ready AND NOT DerotatorControl.Calibrated;
END_IF

// start calibration of focus after elevation has been calibrated
// this avoids imbalance by the M2 mirror on the elvation during its calibration
IF ElevationControl.Calibrated AND NOT FocusControl.Calibrated THEN
	FocusControl.enable := TRUE;
	FocusControl.HomeAxis := TRUE;
END_IF

IF CoverControl.isopen AND 
	ElevationControl.Calibrated AND
	AzimuthElevationControl.calibrated AND
	DerotatorControl.Calibrated AND
	FocusControl.Calibrated THEN
	power := FALSE;
	poweron := TRUE;
	isparked := FALSE;
	// slew the telescope to the home position
	gohome := TRUE;
ELSE
	poweron := FALSE;
END_IF
END_METHOD

METHOD slewtelescope : USINT
VAR_INPUT
END_VAR
VAR
	SlewEvent:	FB_Eventlog;
	command_timeout: TON;
END_VAR
VAR_STAT
	Stage:		USINT := 0;
	LastStage:	USINT := 101;
END_VAR
slewtelescope := Stage;
command_timeout(IN := Stage < 100, PT := T#600S);
IF command_timeout.Q THEN
	error := TRUE;
	errorid := 16#40;
	slew := FALSE;
	Stage := 0;
END_IF
IF reset OR error THEN
	Stage := 0;
END_IF
CASE Stage OF
	0:	
		IF ready AND stopped AND NOT busy AND NOT tracking THEN
			Stage := 25;
		END_IF
	25:
		ElevationControl.position := elevation;
		ElevationControl.velocity := 10.0;
		ElevationControl.MoveAxis := TRUE;
		AzimuthElevationControl.position := azimuth;
		AzimuthElevationControl.velocity := 10.0;
		AzimuthElevationControl.MoveAxis := TRUE;
		DerotatorControl.position := elevation + derotator_offset;
		DerotatorControl.Velocity := 10.0;
		DerotatorControl.MoveAxis := TRUE;
		IF ElevationControl.ElevationAxis.Busy AND
			AzimuthElevationControl.AzimuthAxis.Busy AND
			DerotatorControl.DerotatorAxis.Busy THEN
				Stage := 50;
		END_IF
	50:
		IF ElevationControl.ElevationAxis.MoveDone THEN
			ElevationControl.MoveAxis := FALSE;
		END_IF
		
		IF AzimuthElevationControl.AzimuthAxis.MoveDone THEN
			AzimuthElevationControl.MoveAxis := FALSE;
		END_IF

		IF DerotatorControl.DerotatorAxis.MoveDone THEN
			DerotatorControl.MoveAxis := FALSE;
		END_IF
		IF NOT sliding AND stopped THEN // all axis standstill
			Stage := 100;
		END_IF
	100:
		ElevationControl.MoveAxis := FALSE;
		AzimuthElevationControl.MoveAxis := FALSE;
		DerotatorControl.MoveAxis := FALSE;
		rightascension := rightascension_calc;
		declination := declination_calc;
		slew := FALSE;
		Stage := 0;
END_CASE
SlewEvent(Trigger := Stage > LastStage, FormatString := 'Slew progress: %s', OnMessage := USINT_TO_STRING(Stage));
LastStage := Stage;
END_METHOD

METHOD stoptelescope : BOOL
VAR_INPUT
END_VAR
ElevationControl.StopAxis := TRUE;
AzimuthElevationControl.StopAxis := TRUE;
DerotatorControl.StopAxis := TRUE;
IF stopped THEN
	ElevationControl.StopAxis := FALSE;
	AzimuthElevationControl.StopAxis := FALSE;
	DerotatorControl.StopAxis := FALSE;
	stop := FALSE;
END_IF
END_METHOD

METHOD tracktelescope : BOOL
VAR_INPUT
END_VAR
// Elevation
DerotatorVelocity := F_Derotatorvelocity(elevation_calc, azimuth_calc, latitude);
ElevationVelocity := F_Elevationvelocity(azimuth_calc, latitude);
AzimuthVelocity := F_Azimuthvelocity(elevation_calc, azimuth_calc, latitude);
IF elevation_current < 5.0 OR elevation_current > 89.5 THEN 
	track := FALSE;
END_IF
IF azimuth_current > 440.0 THEN
	track := FALSE;
END_IF
IF (derotator_current < -69.0 AND DerotatorVelocity<0.0) OR (derotator_current > 379.0 AND DerotatorVelocity>0.0) THEN
	track := FALSE;
END_IF

ElevationControl.position := elevation_calc;
IF NOT ElevationControl.Tracking THEN
	ElevationControl.velocity := 10.0;
	ElevationControl.MoveAxis := TRUE;
	IF NOT ElevationControl.ElevationAxis.Busy AND ElevationControl.ElevationAxis.MoveDone THEN
		ElevationControl.MoveAxis := FALSE;
		IF ElevationControl.ElevationAxis.isTracking THEN
			ElevationControl.velocity := ElevationVelocity;
		ELSE
			ElevationControl.velocity := 3.0*ElevationVelocity;
		END_IF
		ElevationControl.velocity := ElevationVelocity;
		ElevationControl.Tracking := TRUE;
	END_IF
ELSE
	ElevationControl.velocity := ElevationVelocity;
END_IF

// Azimuth
AzimuthElevationControl.position := azimuth_calc;
IF NOT AzimuthElevationControl.Tracking THEN
	AzimuthElevationControl.velocity := 10.0;
	AzimuthElevationControl.MoveAxis := TRUE;
	IF NOT AzimuthElevationControl.AzimuthAxis.Busy AND AzimuthElevationControl.AzimuthAxis.MoveDone THEN
		AzimuthElevationControl.MoveAxis := FALSE;
		IF AzimuthElevationControl.AzimuthAxis.isTracking THEN
			AzimuthElevationControl.velocity := AzimuthVelocity;
		ELSE
			AzimuthElevationControl.velocity := 3.0*AzimuthVelocity;
		END_IF
		AzimuthElevationControl.velocity := AzimuthVelocity;
		AzimuthElevationControl.Tracking := TRUE;
	END_IF
ELSE
	AzimuthElevationControl.velocity := AzimuthVelocity;
END_IF

// Derotator
DerotatorControl.position := derotation_calc;
IF NOT DerotatorControl.Tracking THEN
	DerotatorControl.Velocity := 10.0;
	DerotatorControl.MoveAxis := TRUE;
	IF NOT DerotatorControl.DerotatorAxis.Busy AND DerotatorControl.DerotatorAxis.MoveDone THEN
		DerotatorControl.MoveAxis := FALSE;
		IF DerotatorControl.DerotatorAxis.isTracking THEN
			DerotatorControl.Velocity := DerotatorVelocity;
		ELSE
			DerotatorControl.Velocity := 3.0*DerotatorVelocity;
		END_IF
		DerotatorControl.Velocity := DerotatorVelocity;
		DerotatorControl.Tracking := TRUE;
	END_IF
ELSE
	DerotatorControl.Velocity := DerotatorVelocity;
END_IF
END_METHOD

END_PROGRAM

// ---- POUs/TelescopeAuxiliary.TcPOU
PROGRAM TelescopeAuxiliary
VAR
	MQTTTimer : TON := (PT:=T#5S);
END_VAR
VAR_OUTPUT
	// BT9 mirror
	temperature_mirror2:	REAL;
	// BT10
	temperature_mirror1:	REAL;
END_VAR

temperature_mirror1 := GVL_Telescope.temperature_mirror1 / 1000.0;
temperature_mirror2 := GVL_Telescope.temperature_mirror2 / 1000.0;

MQTTTimer(IN:=TRUE);
IF MQTTTimer.Q THEN // publish new payload every second

	MAIN.MQTTClient.Publish('telescope', 'dome', 'Mirror1Temperature',	LREAL_TO_FMTSTR(temperature_mirror1, 2, TRUE));
	MAIN.MQTTClient.Publish('telescope', 'dome', 'Mirror2Temperature',	LREAL_TO_FMTSTR(temperature_mirror2, 2, TRUE));
	
	MQTTTimer(IN:=FALSE);

END_IF

END_PROGRAM

// ---- POUs/MAIN.TcPOU
PROGRAM MAIN
VAR
	// telescope drives are ready to enable
	ready:				BOOL;
	// error stat on drive, power or hydraulics
	error:				BOOL;
	// manual, panel or remote reset
	reset:				BOOL;
	// start hydraulics
	start:				BOOL;
	// stop hydraulics 
	stop:				BOOL;
	// soft start trafo
	key_switch:			BOOL;
	//	open brake
	brake_clearing:		BOOL := FALSE;
	
	remote_start:		BOOL;
	remote_stop: 		BOOL;
	remote_reset:		BOOL;
	remote_keyswitch:	BOOL;
	remote_brake_clearing:	BOOL;
	// blink error lamp on warning
	error_lamp: 		FB_BLINK;
	power_lamp:			FB_BLINK;
	sound_horn:			FB_Horn;
	// main cabinet temperature in degrees
	cabinet_temperature:	REAL;
	TemperatureEvent,
	TemperatureCriticalEvent:	FB_EventLog;
	MQTTTimer : 		TON := (PT:=T#5S);
	GetHostName:		FB_GetHostName;
	HostName: 			STRING(255);
//	LightSwitch:		FB_ButtonEnable;
//	Lightbutton: 		BOOL;
	bExecute:			BOOL := TRUE;
	cabinet_temperature_warning:	SR;
	cabinet_temperature_critical:	SR;
	MQTTClient:		FB_MQTTCommunication;
END_VAR

(* 
Main control loop
* Execute sub modules
* power management
* control panel switches and status lamps

* start switch activates Hydraulics and Trafo
* 
*)
GetHostName(bExecute := bExecute, sHostName => HostName);
bExecute := FALSE;
start := GVL_Main.start_switch OR remote_start;
stop := (NOT GVL_Main.stop_switch) OR remote_stop;
key_switch := GVL_Main.key_switch_remote OR remote_keyswitch;
brake_clearing := GVL_Main.brake_clearing OR remote_brake_clearing;
reset := GVL_Main.reset_switch OR GVL_pendant_control.reset_switch OR remote_reset;		
brake_clearing := NOT GVL_Main.brake_clearing;
cabinet_temperature := INT_TO_REAL(GVL_Main.main_cabinet_temperature) / 10.0;
cabinet_temperature_warning(SET1 := cabinet_temperature > 50.0,
							RESET := cabinet_temperature < 40.0);
cabinet_temperature_critical(SET1 := cabinet_temperature > 60.0,
							RESET := cabinet_temperature < 50.0);

IF start THEN
	HydraulicsControl.enable := TRUE;
END_IF
IF stop THEN
	HydraulicsControl.enable := FALSE;
END_IF

// telescope is ready when power available
ready :=  TRUE;

// QUINT UPS control section
(*
ups(
	xActivate:= xActivate, 
	arrInputPD:= arrInputPD, 
	xActive=> , 
	xError=> , 
	wDiagCode=> , 
	wAddDiagCode=> , 
	wOutputVoltage=> ups_output_voltage, 
	wOutputCurrent=> ups_output_current, 
	xBatModeActive=> , 
	udtDataStruct=> , 
	xAlarm=> , 
	xWarning=> , 
	xReplaceBattery=> , 
	udtDiag=> );
	
ups_output_voltage := ups_output_voltage / 1000.0;
ups_output_current := ups_output_current / 1000.0;
ups_output_power := ups_output_voltage * ups_output_current;
*)

TelescopeControl();	//
CoverControl();	//
PendantControl();	//
HydraulicsControl();	//
ElevationControl();	//
AzimuthElevationControl();	//
DerotatorControl();	//
FocusControl();
//RoofControl();
MQTTClient();
Transformer();

error := GVL_Telescope.azimut_limit_switch
			OR Focuscontrol.Error
			OR CoverControl.Error;
//error := FALSE; // Todo: remove
// set control lights					
GVL_Main.lamp_on_manual := PendantControl.manual;

IF GVL_Safety.Error THEN
	error_lamp.blink := e_blink.short;
ELSIF ElevationControl.error OR AzimuthElevationControl.error OR DerotatorControl.Error THEN
	error_lamp.blink := e_blink.long;
ELSIF HydraulicsControl.oil_warning OR HydraulicsControl.oil_hot OR HydraulicsControl.pressure_failure THEN
	error_lamp.blink := e_blink.slow;
ELSIF error THEN
	error_lamp.blink := e_blink.on;
ELSE
	error_lamp.blink := e_blink.off; 
END_IF

power_lamp.blink := e_blink.on;
error_lamp(Q => GVL_Main.lamp_error);
//GVL_Main.lamp_error := error_lamp.Q;
power_lamp(Q => GVL_Main.lamp_power);
//GVL_Main.lamp_power := power_lamp.Q;

IF GVL_Telescope.azimut_limit_switch THEN
	sound_horn.horn := E_horn.long;
ELSIF Hydraulicscontrol.suction_failure THEN
	sound_horn.horn := E_horn.long;
ELSIF TelescopeControl.poweronwarning.Q THEN
	sound_horn.horn := E_horn.short;
ELSIF Pendantcontrol.horn THEN
	sound_horn.horn := E_horn.beep;
ELSE
	sound_horn.horn := E_horn.off;
END_IF 

sound_horn(Q => GVL_Telescope.horn );

SafetyHandling();

MQTTTimer(IN:=TRUE);
IF MQTTTimer.Q THEN // publish new payload every second
	MQTTTimer(IN:=FALSE);
	MQTTClient.Publish('electronics', 'base', 'MainCabinetTemperature', LREAL_TO_FMTSTR(cabinet_temperature, 2, TRUE));
	MQTTClient.Publish('electronics', 'base', 'MainReady', BOOL_TO_STRING(ready));
	MQTTClient.Publish('electronics', 'base', 'MasterError', BOOL_TO_STRING(error));
END_IF


TemperatureEvent(	
	Trigger := 		cabinet_temperature_warning.Q1, 
	Level := 		ADSLOG_MSGTYPE_WARN,
	FormatString :=	'Main cabinet temperature warning:	%s',
	OnMessage := 	LREAL_TO_FMTSTR( cabinet_temperature, 1, TRUE),);
TemperatureCriticalEvent(	
	Trigger := 		cabinet_temperature_critical.Q1, 
	Level := 		ADSLOG_MSGTYPE_ERROR,
	FormatString :=	'Main cabinet temperature is critical:	%s!',
	OnMessage := 	LREAL_TO_FMTSTR( cabinet_temperature, 1, TRUE),);

END_PROGRAM

// ---- POUs/FunctionBlocks/FB_MQTTCommunication.TcPOU
FUNCTION_BLOCK FB_MQTTCommunication
VAR_INPUT
END_VAR
VAR_OUTPUT
END_VAR
VAR
	GetHostName:		FB_GetHostName;
	HostName: 			STRING(255);
    bSetParameter:		BOOL := FALSE;
    bConnect:			BOOL := FALSE;
    (* received message *)
	bSubscribed: 		BOOL;
	sTopicSub: 			STRING(255) := 'MONETN/Telescope/SET';
	{attribute 'TcEncoding':='UTF-8'}
	sTopicRcv: 			STRING(255);
	{attribute 'TcEncoding':='UTF-8'}
	fbMessageQueue:		FB_IotMqttMessageQueue;
    fbMessage:			FB_IotMqttMessage;
	fbMqttClient:		FB_IotMqttClient;
	sPayloadRcv: 		STRING;
	influxMessage:		FB_InfluxMessage;
	measurement, 
	parameter, 
	value:		STRING(255);
END_VAR

(*
MQTT Communication section

Source:
https://infosys.beckhoff.com/english.php?content=../content/1033/tf6701_tc3_iot_communication_mqtt/3518541195.html&id=

*)
IF HostName='' THEN
	GetHostName.bExecute := TRUE;
ELSE
	GetHostName.bExecute := FALSE;
	bSetParameter := TRUE;
END_IF

GetHostName(sHostName => HostName);

// set the parameters once
IF bSetParameter THEN
    bSetParameter               := FALSE;
    fbMqttClient.sHostName      := '169.254.146.10';
    fbMqttClient.nHostPort      := 1883;
    fbMqttClient.sClientId      := HostName; 
    fbMqttClient.sTopicPrefix   := ''; 
	fbMqttClient.nKeepAlive     := 60; 
    fbMqttClient.ipMessageQueue := fbMessageQueue;
	bConnect := TRUE;
END_IF

// connect to the client
IF NOT fbMqttClient.bConnected THEN
;
END_IF

fbMqttClient.Execute(bConnect);
	
IF fbMqttClient.bConnected THEN
    IF NOT bSubscribed THEN
        bSubscribed := fbMqttClient.Subscribe(sTopic:=sTopicSub, 
												eQoS:=TcIotMqttQos.AtMostOnceDelivery);
    END_IF
END_IF

// receive queued messages
IF fbMessageQueue.nQueuedMessages > 0 THEN
    IF fbMessageQueue.Dequeue(fbMessage:=fbMessage) THEN
        fbMessage.GetTopic(pTopic:=ADR(sTopicRcv), nTopicSize:=SIZEOF(sTopicRcv) );
        fbMessage.GetPayload(pPayload:=ADR(sPayloadRcv), nPayloadSize:=SIZEOF(sPayloadRcv), bSetNullTermination:=TRUE);
		ADSLOGSTR( ADSLOG_MSGTYPE_HINT OR ADSLOG_MSGTYPE_LOG, 'MQTT %s', sPayloadRcv);
		IF sTopicRcv = sTopicSub THEN
			influxMessage(  sPayload := sPayloadRcv, measurement => measurement, parameter => parameter, value => value);
			IF NOT PendantControl.manual AND measurement = 'command' THEN
				IF parameter = 'power' THEN
					TelescopeControl.power := STRING_TO_BOOL(value);
				ELSIF parameter = 'park' THEN
					TelescopeControl.park := STRING_TO_BOOL(value);
				ELSIF parameter = 'gohome' THEN
					TelescopeControl.gohome := STRING_TO_BOOL(value);
				ELSIF parameter = 'track' THEN
					TelescopeControl.track := STRING_TO_BOOL(value);
				ELSIF parameter = 'goto' THEN
					TelescopeControl.goto := STRING_TO_BOOL(value);
				ELSIF parameter = 'slew' THEN
					TelescopeControl.slew := STRING_TO_BOOL(value);
				ELSIF parameter = 'stop' THEN
					TelescopeControl.stop := STRING_TO_BOOL(value);
				ELSIF parameter = 'reset' THEN
					TelescopeControl.reset := STRING_TO_BOOL(value);
				ELSIF parameter = 'masterreset' THEN
					ElevationControl.bSoEReset := STRING_TO_BOOL(value);
					AzimuthElevationControl.bSoEReset := STRING_TO_BOOL(value);
					DerotatorControl.bSoEReset := STRING_TO_BOOL(value);
				ELSIF parameter = 'rightascension' THEN
					TelescopeControl.track := FALSE;
					TelescopeControl.rightascension := STRING_TO_LREAL(value);
				ELSIF parameter = 'declination' THEN
					TelescopeControl.track := FALSE;
					TelescopeControl.declination := STRING_TO_LREAL(value);
				ELSIF parameter = 'elevation' THEN
					TelescopeControl.elevation := STRING_TO_LREAL(value);
				ELSIF parameter = 'azimuth' THEN
					TelescopeControl.azimuth := STRING_TO_LREAL(value);
				ELSIF parameter = 'focus' THEN
					FocusControl.position := STRING_TO_LREAL(value);
				ELSIF parameter = 'derotator' THEN
					TelescopeControl.track := FALSE;
					TelescopeControl.derotator_offset := STRING_TO_LREAL(value);
				ELSIF parameter = 'elevationoffset' THEN
					TelescopeControl.elevation_offset := STRING_TO_LREAL(value);
				ELSIF parameter = 'azimuthoffset' THEN
					TelescopeControl.azimuth_offset := STRING_TO_LREAL(value);
				ELSIF parameter = 'derotatoroffset' THEN
					TelescopeControl.derotator_offset := STRING_TO_LREAL(value);ELSE
					ADSLOGSTR( ADSLOG_MSGTYPE_WARN OR ADSLOG_MSGTYPE_LOG, 'MQTT not understood %s', sPayloadRcv);
				END_IF
			END_IF // measurement
		END_IF // Topic
		sPayloadRcv := '';
    END_IF // Dequeue
END_IF

PROPERTY Error : BOOL
GET
Error := fbMqttClient.bError;
END_GET
END_PROPERTY

METHOD Publish : BOOL
VAR_INPUT
	domain: 	STRING(255) := 'environment';
	location: 	STRING(255) := 'roof';
	parameter:	STRING(255);
	value:		STRING(255);
END_VAR
VAR
	sPayloadPub: STRING(255) := '';
	fbFormat:	FB_FormatString;
	bError:		BOOL;
	nErrID: UDINT;
	retain_message:		BOOL := FALSE;
END_VAR
//sPayloadPub := 'environment,location=roof,host=CX-4E6032 ';
fbFormat( sFormat := '%s,location=%s,host=%s %s=%s', 
			arg1 := F_STRING(domain), 
			arg2 := F_STRING(location), 
			arg3 := F_STRING(HostName),
			arg4 := F_STRING(parameter),
			arg5 := F_STRING(value),
 
			sOut => sPayloadPub,
			bError => bError, 
			nErrID => nErrID );
// retain message if value is boolean
retain_message := value = 'TRUE' OR value = 'FALSE';

Publish := fbMqttClient.Publish(	
				sTopic:= 'MONETN/Telemetry', 
				pPayload:= ADR(sPayloadPub), 
				nPayloadSize:= LEN2(ADR(sPayloadPub)),
				eQoS:= TcIotMqttQos.AtMostOnceDelivery,
				bRetain:= retain_message, 
				bQueue:= FALSE );
END_METHOD

METHOD PublishLog : BOOL
VAR_INPUT
	level: 	STRING(255) := 'INFO';
	message:	STRING(255);
	
END_VAR
VAR
	sPayloadPub: STRING(255) := '';
	fbFormat:	FB_FormatString;
	bError:		BOOL;
	nErrID: UDINT;
END_VAR
VAR_OUTPUT
	published: BOOL;
END_VAR
//sPayloadPub := 'environment,location=roof,host=CX-4E6032 ';
fbFormat( sFormat := 'log,host=%s,level=%s message="%s"', 
			arg1 := F_STRING(HostName), 
			arg2 := F_STRING(level), 
			arg3 := F_STRING(message),
 
			sOut => sPayloadPub,
			bError => bError, 
			nErrID => nErrID );

published := fbMqttClient.Publish(	
				sTopic:= 'MONETN/Log', 
				pPayload:= ADR(sPayloadPub), 
				nPayloadSize:= LEN2(ADR(sPayloadPub)),
				eQoS:= TcIotMqttQos.AtMostOnceDelivery,
				bRetain:= FALSE, 
				bQueue:= FALSE );
END_METHOD

END_FUNCTION_BLOCK

// ---- POUs/HydraulicsControl.TcPOU
PROGRAM HydraulicsControl
VAR_INPUT
	// start the hydraulics
	enable:		BOOL := FALSE;
	// reset any hydraulics error
	reset: 		BOOL;
	// manual override to start the suction pump
	suction_manual:	BOOL;
	//manual override to stop the pump
	pump_manual_stop: BOOL;
END_VAR
VAR_OUTPUT
	// status of the brake: is the brake open?
	brake_open:			BOOL;
	// is the brake closed?
	brake_closed:		BOOL;
	// pump is running, but the pressure remains low
	pressure_failure:	BOOL;
	// suction was started, but it is not running
	suction_failure:	BOOL;
	// main pump is running but suction has a timeout
	hydraulics_failure:	BOOL;
	main_pump_failure: BOOL;
	// oil is low
	oil_low:			BOOL;
	// oil is high (unused?)
	oil_high:			BOOL;
	// oil pressure is 25 bars
	oil_pressure_OK:	BOOL;
	// oil is on reserve
	oil_warning:		BOOL;
	// oil filter is dirty
	oil_filter_dirty:	BOOL;
	// oil is below 10°C
	oil_cold:			BOOL;
	// oil is above 50°C
	oil_hot:			BOOL;
	// main pump is running
	pump_running:		BOOL;
	// suction pump is running
	suction_running :	BOOL := FALSE;
	// error condition
	error: 				BOOL;
END_VAR
VAR
	// command to open the brake
	iopen_brake:	BOOL := FALSE;
	// command to open the brake
	iclose_brake: BOOL;
	// monitors the pressure of the pump is running
	pressure_watchdog:	TON;
	// monitors the activation of the suction pump
	suction_watchdog: TON;
	// monitors the activation of the main pump
	main_pump_watchdog:	TON;
	// watch the hydraulics and suction pumps
	hydraulics_watchdog: TON;
	// the suction pump is activated for at least 55s when maximum is reached
	suction_pump_timer: TOF;
	// represents the state of the main pump
	oil_pump_state:		RS;
	// represents the state of the brake
	brake_state: 		RS;
	// wait for the brake to open after pressure has been established
	brake_open_delay:	TON;
	// report brake opend after a short delay
	brake_opened_delay:	TON;
	// error state (set dominant)
	error_state:	SR;
	// timer to shut off hydraulics after break was closed
	hydraulics_off_timer:	TOF  := (PT := T#30S);
	off_trigger:	F_TRIG;
	HydraulicsLog,
	PumpLog,
	ReserveLog,
	oil_low_log,
	FilterLog,
	OverTemperatureLog,
	UnderTemperatureLog,
	SuctionLog,
	BrakeClearingWarning,
	BrakeHydraulicsWarning,
	BrakeWarning: FB_EventLog;
	
	// measures the operating cycle of the suction pump
	suction_timer : FB_Timer;
	StatusWord, LastStatus:	UDINT;
END_VAR

(* 
Main control Logic for the Hydraulics system
* power on delay for main pump and suction pump
* start main pump if main control is ready (button pressed or remote)
* start suction pump if maximum in pan is reached
* suction pump runs for 60 seconds
* stop main pump if oil is low
* stop main pump if pressure fails for 10 seconds
*)
oil_low := NOT GVL_Hydraulics.oil_low;
oil_high := NOT GVL_Hydraulics.oil_high;
oil_warning := GVL_Hydraulics.oil_reserve;
oil_pressure_OK := GVL_Hydraulics.oil_pressure_OK;
oil_filter_dirty := NOT GVL_Hydraulics.oilfilter_dirty;
oil_cold := NOT GVL_Hydraulics.oil_undertemperature;
oil_hot := GVL_Hydraulics.oil_overtemperature;
pump_running := GVL_Hydraulics.pump_running;
suction_running := GVL_Hydraulics.suction_running;

error_state(SET1 := pressure_failure OR	suction_failure OR hydraulics_failure OR oil_low OR main_pump_failure,
			RESET := reset,
			Q1 => error);

oil_pump_state(SET := enable,
				RESET1 := NOT enable OR error OR pump_manual_stop);

GVL_Hydraulics.oil_pump_enable := oil_pump_state.Q1;

(* This section controls the hydraulic brake responsible for azimuth and elevation. 
Especially the elevation is imbalanced if not in the position control loop. 
The brake must only be opened, if the elevation drive is activated concurrently.
*)


// close the brake if the pump is not running	
IF iclose_brake OR NOT pump_running THEN 
	iopen_brake := FALSE;
END_IF

// wait for pressure to build up (hack for oil_pressure_ok)
brake_open_delay(IN := pump_running AND oil_pressure_OK,
				PT := T#3S);
		
brake_state(SET := brake_open_delay.Q AND iopen_brake AND MAIN.brake_clearing,
			RESET1 := GVL_Telescope.azimut_limit_switch 
					  OR iclose_brake 
					  OR NOT pump_running
					  OR NOT MAIN.brake_clearing,
			Q1 => GVL_Telescope.brake_azimuth_eve);

// signal that the brake is open after one second
brake_opened_delay(	IN :=brake_state.Q1, 
					PT := T#1000MS,
					Q => brake_open);

brake_closed := NOT brake_open;
IF brake_closed THEN
	iclose_brake := FALSE;
END_IF
// turn off the hydraulics if the brake is closed and the pump is still running
hydraulics_off_timer(IN := brake_open AND pump_running );
off_trigger(CLK := hydraulics_off_timer.Q);

IF off_trigger.Q THEN
	enable := FALSE;
END_IF

(* This is the end of the brake control section *)

// measure suction pump cycle
suction_timer(	bStart := suction_running AND NOT suction_pump_timer.Q, 
				bStop := GVL_Hydraulics.oilpan_maximum);  

suction_pump_timer(IN := GVL_Hydraulics.oilpan_maximum,
					PT := T#90S,
					Q => GVL_Hydraulics.oil_suction_enable);
GVL_Hydraulics.oil_suction_enable := suction_pump_timer.Q OR suction_manual;					
suction_watchdog(IN := GVL_Hydraulics.oil_suction_enable AND NOT suction_running,
					PT := T#10S,
					Q => suction_failure);
					
pressure_watchdog(IN := GVL_Hydraulics.oil_pump_enable AND 
						NOT oil_pressure_OK,
					PT := T#30S,
				  Q => pressure_failure);
hydraulics_watchdog(IN := pump_running AND NOT suction_running,
						PT := T#140S,
						Q => hydraulics_failure);

main_pump_watchdog(IN := GVL_Hydraulics.oil_pump_enable AND NOT pump_running,
					PT := T#10S,
					Q => main_pump_failure);

StatusWord.0 := oil_low;
StatusWord.1 := oil_high;
StatusWord.2 := oil_warning;
StatusWord.3 := oil_pressure_OK;
StatusWord.4 := oil_filter_dirty;
StatusWord.5 := oil_cold;
StatusWord.6 := oil_hot;
StatusWord.7 := brake_open;
StatusWord.8 := GVL_Main.brake_clearing;
StatusWord.9 := pump_running;
StatusWord.10 := suction_running;

IF StatusWord<>LastStatus THEN // publish new payload every second
	LastStatus := StatusWord;
	MAIN.MQTTClient.Publish('hydraulics', 'base', 'OilLow',			BOOL_TO_STRING(oil_low));
	MAIN.MQTTClient.Publish('hydraulics', 'base', 'OilHigh',		BOOL_TO_STRING(oil_high));
	MAIN.MQTTClient.Publish('hydraulics', 'base', 'OilReserve',		BOOL_TO_STRING(oil_warning));
	MAIN.MQTTClient.Publish('hydraulics', 'base', 'OilPressureOK', 	BOOL_TO_STRING(oil_pressure_OK));
	MAIN.MQTTClient.Publish('hydraulics', 'base', 'OilFilterDirty',	BOOL_TO_STRING(oil_filter_dirty));
	MAIN.MQTTClient.Publish('hydraulics', 'base', 'OilCold',		BOOL_TO_STRING(oil_cold));
	MAIN.MQTTClient.Publish('hydraulics', 'base', 'OilHot',			BOOL_TO_STRING(oil_Hot));
	MAIN.MQTTClient.Publish('hydraulics', 'base', 'BrakeOpen',		BOOL_TO_STRING(brake_open));
	MAIN.MQTTClient.Publish('hydraulics', 'base', 'BrakeClearing',	BOOL_TO_STRING(GVL_Main.brake_clearing));
	MAIN.MQTTClient.Publish('hydraulics', 'base', 'PumpRunning',	BOOL_TO_STRING(pump_running));
	MAIN.MQTTClient.Publish('hydraulics', 'base', 'SuctionRunning',	BOOL_TO_STRING(suction_running));
END_IF


				  				  
HydraulicsLog(Trigger := pressure_failure OR main_pump_failure,
				Level := ADSLOG_MSGTYPE_ERROR,
				FormatString := 'Main hydraulics pump / pressure: %s',
				OnMessage := 'FAILURE',
				OffMessage := 'OK',
				OffLevel := ADSLOG_MSGTYPE_HINT);

PumpLog(Trigger := pump_running,
				Level := ADSLOG_MSGTYPE_HINT,
				FormatString := 'Main hydraulics pump: %s',
				OnMessage := 'START',
				OffMessage := 'STOP',
				OffLevel := ADSLOG_MSGTYPE_HINT);
	
ReserveLog(Trigger := oil_warning,
			Level := ADSLOG_MSGTYPE_WARN,
			FormatString := 'oil reserve: %s',
			OnMessage := 'LOW',
			OffMessage := 'OK',
			OffLevel := ADSLOG_MSGTYPE_HINT);

oil_low_log(Trigger := oil_low,
				Level := ADSLOG_MSGTYPE_ERROR,
				FormatString := 'oil level: %s',
				OnMessage := 'LOW',
				OffMessage := 'OK',
				OffLevel := ADSLOG_MSGTYPE_HINT);

FilterLog(Trigger := oil_filter_dirty,
				Level := ADSLOG_MSGTYPE_WARN,
				FormatString := 'Hydraulics Filter is %s',
				OnMessage := 'dirty.');

OverTemperatureLog(Trigger := oil_hot,
				Level := ADSLOG_MSGTYPE_WARN,
				FormatString := 'Hydraulics Temperature is %s',
				OnMessage := 'high.');
UnderTemperatureLog(Trigger := oil_cold,
				Level := ADSLOG_MSGTYPE_WARN,
				FormatString := 'Hydraulics Temperature is %s',
				OnMessage := 'low.');

SuctionLog(Trigger := suction_failure OR hydraulics_failure,
				Level := ADSLOG_MSGTYPE_ERROR,
				FormatString := 'suction pump: %s',
				OnMessage := 'FAILURE',
				OffMessage := 'OK',
				OffLevel := ADSLOG_MSGTYPE_HINT);

BrakeClearingWarning(Trigger := NOT Main.brake_clearing AND iopen_brake,
				Level := ADSLOG_MSGTYPE_WARN,
				FormatString := '%s',
				OnMessage := 'Cannot open brake without brake clearing.');

BrakeWarning(	Trigger := brake_open,
				Level := ADSLOG_MSGTYPE_WARN,
				FormatString := '%s',
				OnMessage := 'Brake is open.',
				OffMessage := 'Brake is closed.');

BrakeHydraulicsWarning(Trigger := NOT enable AND iopen_brake,
				Level := ADSLOG_MSGTYPE_WARN,
				FormatString := '%s',
				OnMessage := 'Cannot open brake without running hydraulics.');

METHOD close_brake : BOOL
VAR_INPUT
END_VAR
// close the brake
iclose_brake := TRUE;

RETURN(brake_closed);
END_METHOD

METHOD open_brake : BOOL
VAR_INPUT
END_VAR
// start the pump
enable := TRUE;
// open the brake
IF oil_pressure_OK THEN
	iopen_brake := TRUE;
END_IF;
RETURN(brake_open);
END_METHOD

END_PROGRAM

// ---- POUs/SafetyHandling.TcPOU
PROGRAM SafetyHandling
VAR
	state           : INT := 0;            
	// power on delay
	start_delay 	: TON := (PT := T#2S);
	state_delay 	: TON := (PT := T#1S);

	// Safety group
	fbInfoGroup1			:FB_InfoGroup;
	stInfoGroup1	AT%I*	:ST_InfoDataGroup;
	sStateGroup1			:STRING;
	
	// Estop
	fbInfoEStop1			:FB_InfoEStop;
	stInfoEStop1 	AT%I*	:ST_InfoDataFB;
	sStateEStop1			:STRING;
	sDiagEStop1				:STRING;	
	
	// Errack logging
	ErrAckLog		: FB_EventLog;
	// restart logging
	RestartLog		: FB_EventLog;
	// safety logging
	SafetyLog		: FB_EventLog;
	
END_VAR
VAR_OUTPUT
	// error condition
	Error			: BOOL;
	// Emergency_stop engaged
	Emergency_stop	: BOOL;
END_VAR
VAR_INPUT
	// issue a remote restart
	remote_restart:		BOOL;
	// issue a remute run/stop
	remote_run:			BOOL := TRUE;
END_VAR

// Safety is running on start
GVL_Safety.Run := remote_run;

fbInfoGroup1(
	stInfoData	:= stInfoGroup1,
	sState		=> sStateGroup1);

fbInfoEStop1(
	stInfoData	:= stInfoEStop1, 
	sState		=> sStateEStop1, 
	sDiag		=> sDiagEStop1);

(*

// power on delay for Safety RESTART after RUN=1
start_delay(IN := TRUE);

CASE state OF
	0:
	    IF start_delay.Q  THEN
			GVL_Safety.ErrAck := TRUE;
			state := 1;
		END_IF
	1:
		state_delay(IN := TRUE);	
		IF state_delay.Q THEN
			GVL_Safety.ErrAck := FALSE;
			GVL_Safety.Restart := TRUE;
			state := 2;
			state_delay(IN := FALSE);
		END_IF
	2:
		state_delay(IN := TRUE);	
		IF state_delay.Q THEN
			GVL_Safety.Restart := FALSE;
			GVL_Safety.ErrAck := TRUE;
			state := 3;
			state_delay(IN := FALSE);
		END_IF
	3:
		state_delay(IN := TRUE);	
		IF state_delay.Q THEN	
			GVL_Safety.ErrAck := FALSE;
			state := 4;
			state_delay(IN := FALSE);
		END_IF	
END_CASE

// remote restart
IF remote_restart THEN
	state := 0;
	remote_restart := FALSE;
END_IF

